   1:  PR[GP1:91,1] = PR[GP1:90,1] + 67.544;
   1:  PR[GP1:91,2] = PR[GP1:90,2] + 10.988;
   1:L PR[91] 10mm/sec CNT100;
   1:  PR[GP1:91,1] = PR[GP1:90,1] + 66.651;
   1:  PR[GP1:91,2] = PR[GP1:90,2] + 13.399;
   1:L PR[91] 10mm/sec CNT100;
   1:  PR[GP1:91,1] = PR[GP1:90,1] + 62.807;
   1:  PR[GP1:91,2] = PR[GP1:90,2] + 19.885;
   1:L PR[91] 10mm/sec CNT100;
   1:  PR[GP1:91,1] = PR[GP1:90,1] + 60.998;
   1:  PR[GP1:91,2] = PR[GP1:90,2] + 22.693;
   1:L PR[91] 10mm/sec CNT100;
   1:  PR[GP1:91,1] = PR[GP1:90,1] + 58.011;
   1:  PR[GP1:91,2] = PR[GP1:90,2] + 25.595;
   1:L PR[91] 10mm/sec CNT100;
   1:  PR[GP1:91,1] = PR[GP1:90,1] + 53.750;
   1:  PR[GP1:91,2] = PR[GP1:90,2] + 29.133;
   1:L PR[91] 10mm/sec CNT100;
   1:  PR[GP1:91,1] = PR[GP1:90,1] + 49.246;
   1:  PR[GP1:91,2] = PR[GP1:90,2] + 31.887;
   1:L PR[91] 10mm/sec CNT100;
   1:  PR[GP1:91,1] = PR[GP1:90,1] + 46.434;
   1:  PR[GP1:91,2] = PR[GP1:90,2] + 32.929;
   1:L PR[91] 10mm/sec CNT100;
   1:  PR[GP1:91,1] = PR[GP1:90,1] + 40.608;
   1:  PR[GP1:91,2] = PR[GP1:90,2] + 35.037;
   1:L PR[91] 10mm/sec CNT100;
   1:  PR[GP1:91,1] = PR[GP1:90,1] + 38.148;
   1:  PR[GP1:91,2] = PR[GP1:90,2] + 35.345;
   1:L PR[91] 10mm/sec CNT100;
   1:  PR[GP1:91,1] = PR[GP1:90,1] + 32.674;
   1:  PR[GP1:91,2] = PR[GP1:90,2] + 36.121;
   1:L PR[91] 10mm/sec CNT100;
   1:  PR[GP1:91,1] = PR[GP1:90,1] + 32.260;
   1:  PR[GP1:91,2] = PR[GP1:90,2] + 36.160;
   1:L PR[91] 10mm/sec CNT100;
   1:  PR[GP1:91,1] = PR[GP1:90,1] + 24.335;
   1:  PR[GP1:91,2] = PR[GP1:90,2] + 35.633;
   1:L PR[91] 10mm/sec CNT100;
   1:  PR[GP1:91,1] = PR[GP1:90,1] + 23.229;
   1:  PR[GP1:91,2] = PR[GP1:90,2] + 35.372;
   1:L PR[91] 10mm/sec CNT100;
   1:  PR[GP1:91,1] = PR[GP1:90,1] + 15.787;
   1:  PR[GP1:91,2] = PR[GP1:90,2] + 33.232;
   1:L PR[91] 10mm/sec CNT100;
   1:  PR[GP1:91,1] = PR[GP1:90,1] + 9.527;
   1:  PR[GP1:91,2] = PR[GP1:90,2] + 29.856;
   1:L PR[91] 10mm/sec CNT100;
   1:  PR[GP1:91,1] = PR[GP1:90,1] + 5.825;
   1:  PR[GP1:91,2] = PR[GP1:90,2] + 26.845;
   1:L PR[91] 10mm/sec CNT100;
   1:  PR[GP1:91,1] = PR[GP1:90,1] + 2.865;
   1:  PR[GP1:91,2] = PR[GP1:90,2] + 24.238;
   1:L PR[91] 10mm/sec CNT100;
   1:  PR[GP1:91,1] = PR[GP1:90,1] + 0.407;
   1:  PR[GP1:91,2] = PR[GP1:90,2] + 21.240;
   1:L PR[91] 10mm/sec CNT100;
   1:  PR[GP1:91,1] = PR[GP1:90,1] + -0.917;
   1:L PR[91] 10mm/sec CNT100;
   1:  PR[GP1:91,1] = PR[GP1:90,1] + -3.369;
   1:  PR[GP1:91,2] = PR[GP1:90,2] + 24.219;
   1:L PR[91] 10mm/sec CNT100;
   1:  PR[GP1:91,1] = PR[GP1:90,1] + -6.332;
   1:  PR[GP1:91,2] = PR[GP1:90,2] + 26.828;
   1:L PR[91] 10mm/sec CNT100;
   1:  PR[GP1:91,1] = PR[GP1:90,1] + -10.027;
   1:  PR[GP1:91,2] = PR[GP1:90,2] + 29.832;
   1:L PR[91] 10mm/sec CNT100;
   1:  PR[GP1:91,1] = PR[GP1:90,1] + -16.320;
   1:  PR[GP1:91,2] = PR[GP1:90,2] + 33.236;
   1:L PR[91] 10mm/sec CNT100;
   1:  PR[GP1:91,1] = PR[GP1:90,1] + -23.752;
   1:  PR[GP1:91,2] = PR[GP1:90,2] + 35.373;
   1:L PR[91] 10mm/sec CNT100;
   1:  PR[GP1:91,1] = PR[GP1:90,1] + -24.858;
   1:  PR[GP1:91,2] = PR[GP1:90,2] + 35.634;
   1:L PR[91] 10mm/sec CNT100;
   1:  PR[GP1:91,1] = PR[GP1:90,1] + -32.794;
   1:  PR[GP1:91,2] = PR[GP1:90,2] + 36.157;
   1:L PR[91] 10mm/sec CNT100;
   1:  PR[GP1:91,1] = PR[GP1:90,1] + -38.676;
   1:  PR[GP1:91,2] = PR[GP1:90,2] + 35.343;
   1:L PR[91] 10mm/sec CNT100;
   1:  PR[GP1:91,1] = PR[GP1:90,1] + -41.173;
   1:  PR[GP1:91,2] = PR[GP1:90,2] + 35.029;
   1:L PR[91] 10mm/sec CNT100;
   1:  PR[GP1:91,1] = PR[GP1:90,1] + -49.797;
   1:  PR[GP1:91,2] = PR[GP1:90,2] + 31.874;
   1:L PR[91] 10mm/sec CNT100;
   1:  PR[GP1:91,1] = PR[GP1:90,1] + -54.314;
   1:  PR[GP1:91,2] = PR[GP1:90,2] + 29.097;
   1:L PR[91] 10mm/sec CNT100;
   1:  PR[GP1:91,1] = PR[GP1:90,1] + -58.579;
   1:  PR[GP1:91,2] = PR[GP1:90,2] + 25.562;
   1:L PR[91] 10mm/sec CNT100;
   1:  PR[GP1:91,1] = PR[GP1:90,1] + -61.550;
   1:  PR[GP1:91,2] = PR[GP1:90,2] + 22.671;
   1:L PR[91] 10mm/sec CNT100;
   1:  PR[GP1:91,1] = PR[GP1:90,1] + -65.432;
   1:  PR[GP1:91,2] = PR[GP1:90,2] + 16.136;
   1:L PR[91] 10mm/sec CNT100;
   1:  PR[GP1:91,1] = PR[GP1:90,1] + -67.188;
   1:  PR[GP1:91,2] = PR[GP1:90,2] + 13.362;
   1:L PR[91] 10mm/sec CNT100;
   1:  PR[GP1:91,1] = PR[GP1:90,1] + -68.087;
   1:  PR[GP1:91,2] = PR[GP1:90,2] + 10.901;
   1:L PR[91] 10mm/sec CNT100;
   1:  PR[GP1:91,1] = PR[GP1:90,1] + -69.627;
   1:  PR[GP1:91,2] = PR[GP1:90,2] + 2.415;
   1:L PR[91] 10mm/sec CNT100;
   1:  PR[GP1:91,1] = PR[GP1:90,1] + -69.862;
   1:  PR[GP1:91,2] = PR[GP1:90,2] + 0.301;
   1:L PR[91] 10mm/sec CNT100;
   1:  PR[GP1:91,1] = PR[GP1:90,1] + -68.344;
   1:  PR[GP1:91,2] = PR[GP1:90,2] + -7.941;
   1:L PR[91] 10mm/sec CNT100;
   1:  PR[GP1:91,1] = PR[GP1:90,1] + -68.080;
   1:  PR[GP1:91,2] = PR[GP1:90,2] + -10.363;
   1:L PR[91] 10mm/sec CNT100;
   1:  PR[GP1:91,1] = PR[GP1:90,1] + -67.185;
   1:  PR[GP1:91,2] = PR[GP1:90,2] + -12.813;
   1:L PR[91] 10mm/sec CNT100;
   1:  PR[GP1:91,1] = PR[GP1:90,1] + -63.342;
   1:  PR[GP1:91,2] = PR[GP1:90,2] + -19.317;
   1:L PR[91] 10mm/sec CNT100;
   1:  PR[GP1:91,1] = PR[GP1:90,1] + -61.557;
   1:  PR[GP1:91,2] = PR[GP1:90,2] + -22.106;
   1:L PR[91] 10mm/sec CNT100;
   1:  PR[GP1:91,1] = PR[GP1:90,1] + -58.579;
   1:  PR[GP1:91,2] = PR[GP1:90,2] + -25.004;
   1:L PR[91] 10mm/sec CNT100;
   1:  PR[GP1:91,1] = PR[GP1:90,1] + -54.314;
   1:  PR[GP1:91,2] = PR[GP1:90,2] + -28.539;
   1:L PR[91] 10mm/sec CNT100;
   1:  PR[GP1:91,1] = PR[GP1:90,1] + -49.796;
   1:  PR[GP1:91,2] = PR[GP1:90,2] + -31.317;
   1:L PR[91] 10mm/sec CNT100;
   1:  PR[GP1:91,1] = PR[GP1:90,1] + -46.981;
   1:  PR[GP1:91,2] = PR[GP1:90,2] + -32.360;
   1:L PR[91] 10mm/sec CNT100;
   1:  PR[GP1:91,1] = PR[GP1:90,1] + -41.174;
   1:  PR[GP1:91,2] = PR[GP1:90,2] + -34.471;
   1:L PR[91] 10mm/sec CNT100;
   1:  PR[GP1:91,1] = PR[GP1:90,1] + -38.674;
   1:  PR[GP1:91,2] = PR[GP1:90,2] + -34.785;
   1:L PR[91] 10mm/sec CNT100;
   1:  PR[GP1:91,1] = PR[GP1:90,1] + -33.223;
   1:  PR[GP1:91,2] = PR[GP1:90,2] + -35.561;
   1:L PR[91] 10mm/sec CNT100;
   1:  PR[GP1:91,1] = PR[GP1:90,1] + -32.812;
   1:  PR[GP1:91,2] = PR[GP1:90,2] + -35.600;
   1:L PR[91] 10mm/sec CNT100;
   1:  PR[GP1:91,1] = PR[GP1:90,1] + -24.868;
   1:  PR[GP1:91,2] = PR[GP1:90,2] + -35.076;
   1:L PR[91] 10mm/sec CNT100;
   1:  PR[GP1:91,1] = PR[GP1:90,1] + -23.781;
   1:  PR[GP1:91,2] = PR[GP1:90,2] + -34.828;
   1:L PR[91] 10mm/sec CNT100;
   1:  PR[GP1:91,1] = PR[GP1:90,1] + -16.362;
   1:  PR[GP1:91,2] = PR[GP1:90,2] + -32.697;
   1:L PR[91] 10mm/sec CNT100;
   1:  PR[GP1:91,1] = PR[GP1:90,1] + -15.004;
   1:  PR[GP1:91,2] = PR[GP1:90,2] + -31.901;
   1:L PR[91] 10mm/sec CNT100;
   1:  PR[GP1:91,1] = PR[GP1:90,1] + -9.177;
   1:  PR[GP1:91,2] = PR[GP1:90,2] + -28.729;
   1:L PR[91] 10mm/sec CNT100;
   1:  PR[GP1:91,1] = PR[GP1:90,1] + -6.377;
   1:  PR[GP1:91,2] = PR[GP1:90,2] + -26.314;
   1:L PR[91] 10mm/sec CNT100;
   1:  PR[GP1:91,1] = PR[GP1:90,1] + -3.388;
   1:  PR[GP1:91,2] = PR[GP1:90,2] + -23.682;
   1:L PR[91] 10mm/sec CNT100;
   1:  PR[GP1:91,1] = PR[GP1:90,1] + -0.915;
   1:  PR[GP1:91,2] = PR[GP1:90,2] + -20.682;
   1:L PR[91] 10mm/sec CNT100;
   1:  PR[GP1:91,1] = PR[GP1:90,1] + 0.403;
   1:L PR[91] 10mm/sec CNT100;
   1:  PR[GP1:91,1] = PR[GP1:90,1] + 2.658;
   1:  PR[GP1:91,2] = PR[GP1:90,2] + -23.788;
   1:  PR[GP1:91,3] = PR[GP1:90,3] + 47.275;
   1:L PR[91] 10mm/sec CNT100;
   1:  PR[GP1:91,1] = PR[GP1:90,1] + 5.390;
   1:  PR[GP1:91,2] = PR[GP1:90,2] + -26.193;
   1:L PR[91] 10mm/sec CNT100;
   1:  PR[GP1:91,1] = PR[GP1:90,1] + 8.429;
   1:  PR[GP1:91,2] = PR[GP1:90,2] + -28.820;
   1:L PR[91] 10mm/sec CNT100;
   1:  PR[GP1:91,1] = PR[GP1:90,1] + 14.058;
   1:  PR[GP1:91,2] = PR[GP1:90,2] + -31.876;
   1:L PR[91] 10mm/sec CNT100;
   1:  PR[GP1:91,1] = PR[GP1:90,1] + 15.574;
   1:  PR[GP1:91,2] = PR[GP1:90,2] + -32.763;
   1:L PR[91] 10mm/sec CNT100;
   1:  PR[GP1:91,1] = PR[GP1:90,1] + 22.883;
   1:  PR[GP1:91,2] = PR[GP1:90,2] + -34.862;
   1:L PR[91] 10mm/sec CNT100;
   1:  PR[GP1:91,1] = PR[GP1:90,1] + 24.168;
   1:  PR[GP1:91,2] = PR[GP1:90,2] + -35.156;
   1:L PR[91] 10mm/sec CNT100;
   1:  PR[GP1:91,1] = PR[GP1:90,1] + 31.952;
   1:  PR[GP1:91,2] = PR[GP1:90,2] + -35.673;
   1:L PR[91] 10mm/sec CNT100;
   1:  PR[GP1:91,1] = PR[GP1:90,1] + 40.523;
   1:  PR[GP1:91,2] = PR[GP1:90,2] + -34.492;
   1:L PR[91] 10mm/sec CNT100;
   1:  PR[GP1:91,1] = PR[GP1:90,1] + 48.902;
   1:  PR[GP1:91,2] = PR[GP1:90,2] + -31.442;
   1:L PR[91] 10mm/sec CNT100;
   1:  PR[GP1:91,1] = PR[GP1:90,1] + 53.812;
   1:  PR[GP1:91,2] = PR[GP1:90,2] + -28.438;
   1:L PR[91] 10mm/sec CNT100;
   1:  PR[GP1:91,1] = PR[GP1:90,1] + 57.483;
   1:  PR[GP1:91,2] = PR[GP1:90,2] + -25.391;
   1:L PR[91] 10mm/sec CNT100;
   1:  PR[GP1:91,1] = PR[GP1:90,1] + 60.839;
   1:  PR[GP1:91,2] = PR[GP1:90,2] + -22.131;
   1:L PR[91] 10mm/sec CNT100;
   1:  PR[GP1:91,1] = PR[GP1:90,1] + 64.319;
   1:  PR[GP1:91,2] = PR[GP1:90,2] + -16.291;
   1:L PR[91] 10mm/sec CNT100;
   1:  PR[GP1:91,1] = PR[GP1:90,1] + 66.397;
   1:  PR[GP1:91,2] = PR[GP1:90,2] + -13.029;
   1:L PR[91] 10mm/sec CNT100;
   1:  PR[GP1:91,1] = PR[GP1:90,1] + 67.447;
   1:  PR[GP1:91,2] = PR[GP1:90,2] + -10.193;
   1:L PR[91] 10mm/sec CNT100;
   1:  PR[GP1:91,1] = PR[GP1:90,1] + 68.867;
   1:  PR[GP1:91,2] = PR[GP1:90,2] + -2.360;
   1:L PR[91] 10mm/sec CNT100;
   1:  PR[GP1:91,1] = PR[GP1:90,1] + 69.162;
   1:  PR[GP1:91,2] = PR[GP1:90,2] + 0.258;
   1:L PR[91] 10mm/sec CNT100;
   1:  PR[GP1:91,1] = PR[GP1:90,1] + 67.760;
   1:  PR[GP1:91,2] = PR[GP1:90,2] + 7.881;
   1:L PR[91] 10mm/sec CNT100;
   1:  PR[GP1:91,1] = PR[GP1:90,1] + 67.440;
   1:  PR[GP1:91,2] = PR[GP1:90,2] + 10.771;
   1:L PR[91] 10mm/sec CNT100;
   1:  PR[GP1:91,1] = PR[GP1:90,1] + 66.394;
   1:  PR[GP1:91,2] = PR[GP1:90,2] + 13.597;
   1:L PR[91] 10mm/sec CNT100;
   1:  PR[GP1:91,1] = PR[GP1:90,1] + 62.884;
   1:  PR[GP1:91,2] = PR[GP1:90,2] + 19.520;
   1:L PR[91] 10mm/sec CNT100;
   1:  PR[GP1:91,1] = PR[GP1:90,1] + 60.846;
   1:  PR[GP1:91,2] = PR[GP1:90,2] + 22.682;
   1:L PR[91] 10mm/sec CNT100;
   1:  PR[GP1:91,1] = PR[GP1:90,1] + 57.483;
   1:  PR[GP1:91,2] = PR[GP1:90,2] + 25.949;
   1:L PR[91] 10mm/sec CNT100;
   1:  PR[GP1:91,1] = PR[GP1:90,1] + 53.813;
   1:  PR[GP1:91,2] = PR[GP1:90,2] + 28.996;
   1:L PR[91] 10mm/sec CNT100;
   1:  PR[GP1:91,1] = PR[GP1:90,1] + 48.900;
   1:  PR[GP1:91,2] = PR[GP1:90,2] + 32.001;
   1:L PR[91] 10mm/sec CNT100;
   1:  PR[GP1:91,1] = PR[GP1:90,1] + 46.745;
   1:  PR[GP1:91,2] = PR[GP1:90,2] + 32.799;
   1:L PR[91] 10mm/sec CNT100;
   1:  PR[GP1:91,1] = PR[GP1:90,1] + 40.523;
   1:  PR[GP1:91,2] = PR[GP1:90,2] + 35.050;
   1:L PR[91] 10mm/sec CNT100;
   1:  PR[GP1:91,1] = PR[GP1:90,1] + 32.575;
   1:  PR[GP1:91,2] = PR[GP1:90,2] + 36.174;
   1:L PR[91] 10mm/sec CNT100;
   1:  PR[GP1:91,1] = PR[GP1:90,1] + 31.958;
   1:  PR[GP1:91,2] = PR[GP1:90,2] + 36.231;
   1:L PR[91] 10mm/sec CNT100;
   1:  PR[GP1:91,1] = PR[GP1:90,1] + 24.156;
   1:  PR[GP1:91,2] = PR[GP1:90,2] + 35.713;
   1:L PR[91] 10mm/sec CNT100;
   1:  PR[GP1:91,1] = PR[GP1:90,1] + 22.848;
   1:  PR[GP1:91,2] = PR[GP1:90,2] + 35.404;
   1:L PR[91] 10mm/sec CNT100;
   1:  PR[GP1:91,1] = PR[GP1:90,1] + 15.529;
   1:  PR[GP1:91,2] = PR[GP1:90,2] + 33.300;
   1:L PR[91] 10mm/sec CNT100;
   1:  PR[GP1:91,1] = PR[GP1:90,1] + 9.354;
   1:  PR[GP1:91,2] = PR[GP1:90,2] + 29.970;
   1:L PR[91] 10mm/sec CNT100;
   1:  PR[GP1:91,1] = PR[GP1:90,1] + 5.340;
   1:  PR[GP1:91,2] = PR[GP1:90,2] + 26.705;
   1:L PR[91] 10mm/sec CNT100;
   1:  PR[GP1:91,1] = PR[GP1:90,1] + 2.636;
   1:  PR[GP1:91,2] = PR[GP1:90,2] + 24.324;
   1:L PR[91] 10mm/sec CNT100;
   1:  PR[GP1:91,1] = PR[GP1:90,1] + 0.374;
   1:  PR[GP1:91,2] = PR[GP1:90,2] + 21.565;
   1:L PR[91] 10mm/sec CNT100;
   1:  PR[GP1:91,1] = PR[GP1:90,1] + -0.885;
   1:L PR[91] 10mm/sec CNT100;
   1:  PR[GP1:91,1] = PR[GP1:90,1] + -3.142;
   1:  PR[GP1:91,2] = PR[GP1:90,2] + 24.306;
   1:L PR[91] 10mm/sec CNT100;
   1:  PR[GP1:91,1] = PR[GP1:90,1] + -5.849;
   1:  PR[GP1:91,2] = PR[GP1:90,2] + 26.690;
   1:L PR[91] 10mm/sec CNT100;
   1:  PR[GP1:91,1] = PR[GP1:90,1] + -9.854;
   1:  PR[GP1:91,2] = PR[GP1:90,2] + 29.946;
   1:L PR[91] 10mm/sec CNT100;
   1:  PR[GP1:91,1] = PR[GP1:90,1] + -16.062;
   1:  PR[GP1:91,2] = PR[GP1:90,2] + 33.303;
   1:L PR[91] 10mm/sec CNT100;
   1:  PR[GP1:91,1] = PR[GP1:90,1] + -23.371;
   1:  PR[GP1:91,2] = PR[GP1:90,2] + 35.405;
   1:L PR[91] 10mm/sec CNT100;
   1:  PR[GP1:91,1] = PR[GP1:90,1] + -24.679;
   1:  PR[GP1:91,2] = PR[GP1:90,2] + 35.714;
   1:L PR[91] 10mm/sec CNT100;
   1:  PR[GP1:91,1] = PR[GP1:90,1] + -32.492;
   1:  PR[GP1:91,2] = PR[GP1:90,2] + 36.229;
   1:L PR[91] 10mm/sec CNT100;
   1:  PR[GP1:91,1] = PR[GP1:90,1] + -41.091;
   1:  PR[GP1:91,2] = PR[GP1:90,2] + 35.042;
   1:L PR[91] 10mm/sec CNT100;
   1:  PR[GP1:91,1] = PR[GP1:90,1] + -49.453;
   1:  PR[GP1:91,2] = PR[GP1:90,2] + 31.987;
   1:L PR[91] 10mm/sec CNT100;
   1:  PR[GP1:91,1] = PR[GP1:90,1] + -54.380;
   1:  PR[GP1:91,2] = PR[GP1:90,2] + 28.958;
   1:L PR[91] 10mm/sec CNT100;
   1:  PR[GP1:91,1] = PR[GP1:90,1] + -58.056;
   1:  PR[GP1:91,2] = PR[GP1:90,2] + 25.911;
   1:L PR[91] 10mm/sec CNT100;
   1:  PR[GP1:91,1] = PR[GP1:90,1] + -61.402;
   1:  PR[GP1:91,2] = PR[GP1:90,2] + 22.655;
   1:L PR[91] 10mm/sec CNT100;
   1:  PR[GP1:91,1] = PR[GP1:90,1] + -64.883;
   1:  PR[GP1:91,2] = PR[GP1:90,2] + 16.796;
   1:L PR[91] 10mm/sec CNT100;
   1:  PR[GP1:91,1] = PR[GP1:90,1] + -66.932;
   1:  PR[GP1:91,2] = PR[GP1:90,2] + 13.559;
   1:L PR[91] 10mm/sec CNT100;
   1:  PR[GP1:91,1] = PR[GP1:90,1] + -67.986;
   1:  PR[GP1:91,2] = PR[GP1:90,2] + 10.676;
   1:L PR[91] 10mm/sec CNT100;
   1:  PR[GP1:91,1] = PR[GP1:90,1] + -69.404;
   1:  PR[GP1:91,2] = PR[GP1:90,2] + 2.859;
   1:L PR[91] 10mm/sec CNT100;
   1:  PR[GP1:91,1] = PR[GP1:90,1] + -69.689;
   1:  PR[GP1:91,2] = PR[GP1:90,2] + 0.301;
   1:L PR[91] 10mm/sec CNT100;
   1:  PR[GP1:91,1] = PR[GP1:90,1] + -68.287;
   1:  PR[GP1:91,2] = PR[GP1:90,2] + -7.309;
   1:L PR[91] 10mm/sec CNT100;
   1:  PR[GP1:91,1] = PR[GP1:90,1] + -67.978;
   1:  PR[GP1:91,2] = PR[GP1:90,2] + -10.138;
   1:L PR[91] 10mm/sec CNT100;
   1:  PR[GP1:91,1] = PR[GP1:90,1] + -66.929;
   1:  PR[GP1:91,2] = PR[GP1:90,2] + -13.010;
   1:L PR[91] 10mm/sec CNT100;
   1:  PR[GP1:91,1] = PR[GP1:90,1] + -63.419;
   1:  PR[GP1:91,2] = PR[GP1:90,2] + -18.950;
   1:L PR[91] 10mm/sec CNT100;
   1:  PR[GP1:91,1] = PR[GP1:90,1] + -61.409;
   1:  PR[GP1:91,2] = PR[GP1:90,2] + -22.090;
   1:L PR[91] 10mm/sec CNT100;
   1:  PR[GP1:91,1] = PR[GP1:90,1] + -58.056;
   1:  PR[GP1:91,2] = PR[GP1:90,2] + -25.353;
   1:L PR[91] 10mm/sec CNT100;
   1:  PR[GP1:91,1] = PR[GP1:90,1] + -54.380;
   1:  PR[GP1:91,2] = PR[GP1:90,2] + -28.400;
   1:L PR[91] 10mm/sec CNT100;
   1:  PR[GP1:91,1] = PR[GP1:90,1] + -49.452;
   1:  PR[GP1:91,2] = PR[GP1:90,2] + -31.430;
   1:L PR[91] 10mm/sec CNT100;
   1:  PR[GP1:91,1] = PR[GP1:90,1] + -47.293;
   1:  PR[GP1:91,2] = PR[GP1:90,2] + -32.230;
   1:L PR[91] 10mm/sec CNT100;
   1:  PR[GP1:91,1] = PR[GP1:90,1] + -41.091;
   1:  PR[GP1:91,2] = PR[GP1:90,2] + -34.484;
   1:L PR[91] 10mm/sec CNT100;
   1:  PR[GP1:91,1] = PR[GP1:90,1] + -33.126;
   1:  PR[GP1:91,2] = PR[GP1:90,2] + -35.614;
   1:L PR[91] 10mm/sec CNT100;
   1:  PR[GP1:91,1] = PR[GP1:90,1] + -32.512;
   1:  PR[GP1:91,2] = PR[GP1:90,2] + -35.672;
   1:L PR[91] 10mm/sec CNT100;
   1:  PR[GP1:91,1] = PR[GP1:90,1] + -24.691;
   1:  PR[GP1:91,2] = PR[GP1:90,2] + -35.156;
   1:L PR[91] 10mm/sec CNT100;
   1:  PR[GP1:91,1] = PR[GP1:90,1] + -23.406;
   1:  PR[GP1:91,2] = PR[GP1:90,2] + -34.862;
   1:L PR[91] 10mm/sec CNT100;
   1:  PR[GP1:91,1] = PR[GP1:90,1] + -16.107;
   1:  PR[GP1:91,2] = PR[GP1:90,2] + -32.766;
   1:L PR[91] 10mm/sec CNT100;
   1:  PR[GP1:91,1] = PR[GP1:90,1] + -14.593;
   1:  PR[GP1:91,2] = PR[GP1:90,2] + -31.879;
   1:L PR[91] 10mm/sec CNT100;
   1:  PR[GP1:91,1] = PR[GP1:90,1] + -8.933;
   1:  PR[GP1:91,2] = PR[GP1:90,2] + -28.798;
   1:L PR[91] 10mm/sec CNT100;
   1:  PR[GP1:91,1] = PR[GP1:90,1] + -5.897;
   1:  PR[GP1:91,2] = PR[GP1:90,2] + -26.179;
   1:L PR[91] 10mm/sec CNT100;
   1:  PR[GP1:91,1] = PR[GP1:90,1] + -3.162;
   1:  PR[GP1:91,2] = PR[GP1:90,2] + -23.771;
   1:L PR[91] 10mm/sec CNT100;
   1:  PR[GP1:91,1] = PR[GP1:90,1] + -0.884;
   1:  PR[GP1:91,2] = PR[GP1:90,2] + -21.007;
   1:L PR[91] 10mm/sec CNT100;
   1:  PR[GP1:91,1] = PR[GP1:90,1] + 0.371;
   1:L PR[91] 10mm/sec CNT100;
   1:  PR[GP1:91,1] = PR[GP1:90,1] + 2.431;
   1:  PR[GP1:91,2] = PR[GP1:90,2] + -23.875;
   1:  PR[GP1:91,3] = PR[GP1:90,3] + 47.885;
   1:L PR[91] 10mm/sec CNT100;
   1:  PR[GP1:91,1] = PR[GP1:90,1] + 4.909;
   1:  PR[GP1:91,2] = PR[GP1:90,2] + -26.057;
   1:L PR[91] 10mm/sec CNT100;
   1:  PR[GP1:91,1] = PR[GP1:90,1] + 8.185;
   1:  PR[GP1:91,2] = PR[GP1:90,2] + -28.889;
   1:L PR[91] 10mm/sec CNT100;
   1:  PR[GP1:91,1] = PR[GP1:90,1] + 13.648;
   1:  PR[GP1:91,2] = PR[GP1:90,2] + -31.854;
   1:L PR[91] 10mm/sec CNT100;
   1:  PR[GP1:91,1] = PR[GP1:90,1] + 15.319;
   1:  PR[GP1:91,2] = PR[GP1:90,2] + -32.832;
   1:L PR[91] 10mm/sec CNT100;
   1:  PR[GP1:91,1] = PR[GP1:90,1] + 22.507;
   1:  PR[GP1:91,2] = PR[GP1:90,2] + -34.896;
   1:L PR[91] 10mm/sec CNT100;
   1:  PR[GP1:91,1] = PR[GP1:90,1] + 23.991;
   1:  PR[GP1:91,2] = PR[GP1:90,2] + -35.236;
   1:L PR[91] 10mm/sec CNT100;
   1:  PR[GP1:91,1] = PR[GP1:90,1] + 31.652;
   1:  PR[GP1:91,2] = PR[GP1:90,2] + -35.745;
   1:L PR[91] 10mm/sec CNT100;
   1:  PR[GP1:91,1] = PR[GP1:90,1] + 40.318;
   1:  PR[GP1:91,2] = PR[GP1:90,2] + -34.557;
   1:L PR[91] 10mm/sec CNT100;
   1:  PR[GP1:91,1] = PR[GP1:90,1] + 48.556;
   1:  PR[GP1:91,2] = PR[GP1:90,2] + -31.556;
   1:L PR[91] 10mm/sec CNT100;
   1:  PR[GP1:91,1] = PR[GP1:90,1] + 53.875;
   1:  PR[GP1:91,2] = PR[GP1:90,2] + -28.302;
   1:L PR[91] 10mm/sec CNT100;
   1:  PR[GP1:91,1] = PR[GP1:90,1] + 56.955;
   1:  PR[GP1:91,2] = PR[GP1:90,2] + -25.745;
   1:L PR[91] 10mm/sec CNT100;
   1:  PR[GP1:91,1] = PR[GP1:90,1] + 60.687;
   1:  PR[GP1:91,2] = PR[GP1:90,2] + -22.120;
   1:L PR[91] 10mm/sec CNT100;
   1:  PR[GP1:91,1] = PR[GP1:90,1] + 63.765;
   1:  PR[GP1:91,2] = PR[GP1:90,2] + -16.956;
   1:L PR[91] 10mm/sec CNT100;
   1:  PR[GP1:91,1] = PR[GP1:90,1] + 66.140;
   1:  PR[GP1:91,2] = PR[GP1:90,2] + -13.227;
   1:L PR[91] 10mm/sec CNT100;
   1:  PR[GP1:91,1] = PR[GP1:90,1] + 67.344;
   1:  PR[GP1:91,2] = PR[GP1:90,2] + -9.976;
   1:L PR[91] 10mm/sec CNT100;
   1:  PR[GP1:91,1] = PR[GP1:90,1] + 68.641;
   1:  PR[GP1:91,2] = PR[GP1:90,2] + -2.814;
   1:L PR[91] 10mm/sec CNT100;
   1:  PR[GP1:91,1] = PR[GP1:90,1] + 68.988;
   1:  PR[GP1:91,2] = PR[GP1:90,2] + 0.258;
   1:L PR[91] 10mm/sec CNT100;
   1:  PR[GP1:91,1] = PR[GP1:90,1] + 67.703;
   1:  PR[GP1:91,2] = PR[GP1:90,2] + 7.248;
   1:L PR[91] 10mm/sec CNT100;
   1:  PR[GP1:91,1] = PR[GP1:90,1] + 67.337;
   1:  PR[GP1:91,2] = PR[GP1:90,2] + 10.553;
   1:L PR[91] 10mm/sec CNT100;
   1:  PR[GP1:91,1] = PR[GP1:90,1] + 66.136;
   1:  PR[GP1:91,2] = PR[GP1:90,2] + 13.795;
   1:L PR[91] 10mm/sec CNT100;
   1:  PR[GP1:91,1] = PR[GP1:90,1] + 62.960;
   1:  PR[GP1:91,2] = PR[GP1:90,2] + 19.154;
   1:L PR[91] 10mm/sec CNT100;
   1:  PR[GP1:91,1] = PR[GP1:90,1] + 60.695;
   1:  PR[GP1:91,2] = PR[GP1:90,2] + 22.670;
   1:L PR[91] 10mm/sec CNT100;
   1:  PR[GP1:91,1] = PR[GP1:90,1] + 56.955;
   1:  PR[GP1:91,2] = PR[GP1:90,2] + 26.303;
   1:L PR[91] 10mm/sec CNT100;
   1:  PR[GP1:91,1] = PR[GP1:90,1] + 53.875;
   1:  PR[GP1:91,2] = PR[GP1:90,2] + 28.860;
   1:L PR[91] 10mm/sec CNT100;
   1:  PR[GP1:91,1] = PR[GP1:90,1] + 48.556;
   1:  PR[GP1:91,2] = PR[GP1:90,2] + 32.114;
   1:L PR[91] 10mm/sec CNT100;
   1:  PR[GP1:91,1] = PR[GP1:90,1] + 40.315;
   1:  PR[GP1:91,2] = PR[GP1:90,2] + 35.116;
   1:L PR[91] 10mm/sec CNT100;
   1:  PR[GP1:91,1] = PR[GP1:90,1] + 32.476;
   1:  PR[GP1:91,2] = PR[GP1:90,2] + 36.227;
   1:L PR[91] 10mm/sec CNT100;
   1:  PR[GP1:91,1] = PR[GP1:90,1] + 31.655;
   1:  PR[GP1:91,2] = PR[GP1:90,2] + 36.303;
   1:L PR[91] 10mm/sec CNT100;
   1:  PR[GP1:91,1] = PR[GP1:90,1] + 23.977;
   1:  PR[GP1:91,2] = PR[GP1:90,2] + 35.793;
   1:L PR[91] 10mm/sec CNT100;
   1:  PR[GP1:91,1] = PR[GP1:90,1] + 22.468;
   1:  PR[GP1:91,2] = PR[GP1:90,2] + 35.437;
   1:L PR[91] 10mm/sec CNT100;
   1:  PR[GP1:91,1] = PR[GP1:90,1] + 15.271;
   1:  PR[GP1:91,2] = PR[GP1:90,2] + 33.368;
   1:L PR[91] 10mm/sec CNT100;
   1:  PR[GP1:91,1] = PR[GP1:90,1] + 9.182;
   1:  PR[GP1:91,2] = PR[GP1:90,2] + 30.084;
   1:L PR[91] 10mm/sec CNT100;
   1:  PR[GP1:91,1] = PR[GP1:90,1] + 4.855;
   1:  PR[GP1:91,2] = PR[GP1:90,2] + 26.566;
   1:L PR[91] 10mm/sec CNT100;
   1:  PR[GP1:91,1] = PR[GP1:90,1] + 2.407;
   1:  PR[GP1:91,2] = PR[GP1:90,2] + 24.409;
   1:L PR[91] 10mm/sec CNT100;
   1:  PR[GP1:91,1] = PR[GP1:90,1] + 0.341;
   1:  PR[GP1:91,2] = PR[GP1:90,2] + 21.890;
   1:L PR[91] 10mm/sec CNT100;
   1:  PR[GP1:91,1] = PR[GP1:90,1] + -0.854;
   1:L PR[91] 10mm/sec CNT100;
   1:  PR[GP1:91,1] = PR[GP1:90,1] + -2.914;
   1:  PR[GP1:91,2] = PR[GP1:90,2] + 24.393;
   1:L PR[91] 10mm/sec CNT100;
   1:  PR[GP1:91,1] = PR[GP1:90,1] + -5.366;
   1:  PR[GP1:91,2] = PR[GP1:90,2] + 26.552;
   1:L PR[91] 10mm/sec CNT100;
   1:  PR[GP1:91,1] = PR[GP1:90,1] + -9.682;
   1:  PR[GP1:91,2] = PR[GP1:90,2] + 30.061;
   1:L PR[91] 10mm/sec CNT100;
   1:  PR[GP1:91,1] = PR[GP1:90,1] + -15.803;
   1:  PR[GP1:91,2] = PR[GP1:90,2] + 33.371;
   1:L PR[91] 10mm/sec CNT100;
   1:  PR[GP1:91,1] = PR[GP1:90,1] + -22.990;
   1:  PR[GP1:91,2] = PR[GP1:90,2] + 35.437;
   1:L PR[91] 10mm/sec CNT100;
   1:  PR[GP1:91,1] = PR[GP1:90,1] + -24.500;
   1:  PR[GP1:91,2] = PR[GP1:90,2] + 35.794;
   1:L PR[91] 10mm/sec CNT100;
   1:  PR[GP1:91,1] = PR[GP1:90,1] + -32.189;
   1:  PR[GP1:91,2] = PR[GP1:90,2] + 36.301;
   1:L PR[91] 10mm/sec CNT100;
   1:  PR[GP1:91,1] = PR[GP1:90,1] + -40.886;
   1:  PR[GP1:91,2] = PR[GP1:90,2] + 35.106;
   1:L PR[91] 10mm/sec CNT100;
   1:  PR[GP1:91,1] = PR[GP1:90,1] + -49.109;
   1:  PR[GP1:91,2] = PR[GP1:90,2] + 32.100;
   1:L PR[91] 10mm/sec CNT100;
   1:  PR[GP1:91,1] = PR[GP1:90,1] + -54.446;
   1:  PR[GP1:91,2] = PR[GP1:90,2] + 28.819;
   1:L PR[91] 10mm/sec CNT100;
   1:  PR[GP1:91,1] = PR[GP1:90,1] + -57.533;
   1:  PR[GP1:91,2] = PR[GP1:90,2] + 26.260;
   1:L PR[91] 10mm/sec CNT100;
   1:  PR[GP1:91,1] = PR[GP1:90,1] + -61.254;
   1:  PR[GP1:91,2] = PR[GP1:90,2] + 22.640;
   1:L PR[91] 10mm/sec CNT100;
   1:  PR[GP1:91,1] = PR[GP1:90,1] + -64.334;
   1:  PR[GP1:91,2] = PR[GP1:90,2] + 17.456;
   1:L PR[91] 10mm/sec CNT100;
   1:  PR[GP1:91,1] = PR[GP1:90,1] + -66.676;
   1:  PR[GP1:91,2] = PR[GP1:90,2] + 13.756;
   1:L PR[91] 10mm/sec CNT100;
   1:  PR[GP1:91,1] = PR[GP1:90,1] + -67.884;
   1:  PR[GP1:91,2] = PR[GP1:90,2] + 10.450;
   1:L PR[91] 10mm/sec CNT100;
   1:  PR[GP1:91,1] = PR[GP1:90,1] + -69.181;
   1:  PR[GP1:91,2] = PR[GP1:90,2] + 3.302;
   1:L PR[91] 10mm/sec CNT100;
   1:  PR[GP1:91,1] = PR[GP1:90,1] + -69.515;
   1:  PR[GP1:91,2] = PR[GP1:90,2] + 0.301;
   1:L PR[91] 10mm/sec CNT100;
   1:  PR[GP1:91,1] = PR[GP1:90,1] + -68.229;
   1:  PR[GP1:91,2] = PR[GP1:90,2] + -6.678;
   1:L PR[91] 10mm/sec CNT100;
   1:  PR[GP1:91,1] = PR[GP1:90,1] + -67.876;
   1:  PR[GP1:91,2] = PR[GP1:90,2] + -9.912;
   1:L PR[91] 10mm/sec CNT100;
   1:  PR[GP1:91,1] = PR[GP1:90,1] + -66.673;
   1:  PR[GP1:91,2] = PR[GP1:90,2] + -13.206;
   1:L PR[91] 10mm/sec CNT100;
   1:  PR[GP1:91,1] = PR[GP1:90,1] + -63.497;
   1:  PR[GP1:91,2] = PR[GP1:90,2] + -18.582;
   1:L PR[91] 10mm/sec CNT100;
   1:  PR[GP1:91,1] = PR[GP1:90,1] + -61.262;
   1:  PR[GP1:91,2] = PR[GP1:90,2] + -22.074;
   1:L PR[91] 10mm/sec CNT100;
   1:  PR[GP1:91,1] = PR[GP1:90,1] + -57.533;
   1:  PR[GP1:91,2] = PR[GP1:90,2] + -25.702;
   1:L PR[91] 10mm/sec CNT100;
   1:  PR[GP1:91,1] = PR[GP1:90,1] + -54.446;
   1:  PR[GP1:91,2] = PR[GP1:90,2] + -28.261;
   1:L PR[91] 10mm/sec CNT100;
   1:  PR[GP1:91,1] = PR[GP1:90,1] + -49.109;
   1:  PR[GP1:91,2] = PR[GP1:90,2] + -31.542;
   1:L PR[91] 10mm/sec CNT100;
   1:  PR[GP1:91,1] = PR[GP1:90,1] + -40.887;
   1:  PR[GP1:91,2] = PR[GP1:90,2] + -34.548;
   1:L PR[91] 10mm/sec CNT100;
   1:  PR[GP1:91,1] = PR[GP1:90,1] + -33.028;
   1:  PR[GP1:91,2] = PR[GP1:90,2] + -35.666;
   1:L PR[91] 10mm/sec CNT100;
   1:  PR[GP1:91,1] = PR[GP1:90,1] + -32.211;
   1:  PR[GP1:91,2] = PR[GP1:90,2] + -35.744;
   1:L PR[91] 10mm/sec CNT100;
   1:  PR[GP1:91,1] = PR[GP1:90,1] + -24.515;
   1:  PR[GP1:91,2] = PR[GP1:90,2] + -35.237;
   1:L PR[91] 10mm/sec CNT100;
   1:  PR[GP1:91,1] = PR[GP1:90,1] + -23.031;
   1:  PR[GP1:91,2] = PR[GP1:90,2] + -34.897;
   1:L PR[91] 10mm/sec CNT100;
   1:  PR[GP1:91,1] = PR[GP1:90,1] + -15.852;
   1:  PR[GP1:91,2] = PR[GP1:90,2] + -32.836;
   1:L PR[91] 10mm/sec CNT100;
   1:  PR[GP1:91,1] = PR[GP1:90,1] + -14.182;
   1:  PR[GP1:91,2] = PR[GP1:90,2] + -31.857;
   1:L PR[91] 10mm/sec CNT100;
   1:  PR[GP1:91,1] = PR[GP1:90,1] + -8.689;
   1:  PR[GP1:91,2] = PR[GP1:90,2] + -28.867;
   1:L PR[91] 10mm/sec CNT100;
   1:  PR[GP1:91,1] = PR[GP1:90,1] + -5.417;
   1:  PR[GP1:91,2] = PR[GP1:90,2] + -26.044;
   1:L PR[91] 10mm/sec CNT100;
   1:  PR[GP1:91,1] = PR[GP1:90,1] + -2.936;
   1:  PR[GP1:91,2] = PR[GP1:90,2] + -23.859;
   1:L PR[91] 10mm/sec CNT100;
   1:  PR[GP1:91,1] = PR[GP1:90,1] + -0.853;
   1:  PR[GP1:91,2] = PR[GP1:90,2] + -21.332;
   1:L PR[91] 10mm/sec CNT100;
   1:  PR[GP1:91,1] = PR[GP1:90,1] + 0.339;
   1:L PR[91] 10mm/sec CNT100;
   1:  PR[GP1:91,1] = PR[GP1:90,1] + 2.203;
   1:  PR[GP1:91,2] = PR[GP1:90,2] + -23.962;
   1:  PR[GP1:91,3] = PR[GP1:90,3] + 48.495;
   1:L PR[91] 10mm/sec CNT100;
   1:  PR[GP1:91,1] = PR[GP1:90,1] + 4.427;
   1:  PR[GP1:91,2] = PR[GP1:90,2] + -25.921;
   1:L PR[91] 10mm/sec CNT100;
   1:  PR[GP1:91,1] = PR[GP1:90,1] + 7.941;
   1:  PR[GP1:91,2] = PR[GP1:90,2] + -28.957;
   1:L PR[91] 10mm/sec CNT100;
   1:  PR[GP1:91,1] = PR[GP1:90,1] + 13.237;
   1:  PR[GP1:91,2] = PR[GP1:90,2] + -31.832;
   1:L PR[91] 10mm/sec CNT100;
   1:  PR[GP1:91,1] = PR[GP1:90,1] + 15.065;
   1:  PR[GP1:91,2] = PR[GP1:90,2] + -32.902;
   1:L PR[91] 10mm/sec CNT100;
   1:  PR[GP1:91,1] = PR[GP1:90,1] + 22.132;
   1:  PR[GP1:91,2] = PR[GP1:90,2] + -34.931;
   1:L PR[91] 10mm/sec CNT100;
   1:  PR[GP1:91,1] = PR[GP1:90,1] + 23.814;
   1:  PR[GP1:91,2] = PR[GP1:90,2] + -35.316;
   1:L PR[91] 10mm/sec CNT100;
   1:  PR[GP1:91,1] = PR[GP1:90,1] + 31.352;
   1:  PR[GP1:91,2] = PR[GP1:90,2] + -35.817;
   1:L PR[91] 10mm/sec CNT100;
   1:  PR[GP1:91,1] = PR[GP1:90,1] + 39.758;
   1:  PR[GP1:91,2] = PR[GP1:90,2] + -34.657;
   1:L PR[91] 10mm/sec CNT100;
   1:  PR[GP1:91,1] = PR[GP1:90,1] + 40.112;
   1:  PR[GP1:91,2] = PR[GP1:90,2] + -34.622;
   1:L PR[91] 10mm/sec CNT100;
   1:  PR[GP1:91,1] = PR[GP1:90,1] + 48.209;
   1:  PR[GP1:91,2] = PR[GP1:90,2] + -31.670;
   1:L PR[91] 10mm/sec CNT100;
   1:  PR[GP1:91,1] = PR[GP1:90,1] + 53.938;
   1:  PR[GP1:91,2] = PR[GP1:90,2] + -28.166;
   1:L PR[91] 10mm/sec CNT100;
   1:  PR[GP1:91,1] = PR[GP1:90,1] + 56.427;
   1:  PR[GP1:91,2] = PR[GP1:90,2] + -26.099;
   1:L PR[91] 10mm/sec CNT100;
   1:  PR[GP1:91,1] = PR[GP1:90,1] + 60.535;
   1:  PR[GP1:91,2] = PR[GP1:90,2] + -22.108;
   1:L PR[91] 10mm/sec CNT100;
   1:  PR[GP1:91,1] = PR[GP1:90,1] + 63.210;
   1:  PR[GP1:91,2] = PR[GP1:90,2] + -17.621;
   1:L PR[91] 10mm/sec CNT100;
   1:  PR[GP1:91,1] = PR[GP1:90,1] + 65.882;
   1:  PR[GP1:91,2] = PR[GP1:90,2] + -13.425;
   1:L PR[91] 10mm/sec CNT100;
   1:  PR[GP1:91,1] = PR[GP1:90,1] + 67.240;
   1:  PR[GP1:91,2] = PR[GP1:90,2] + -9.758;
   1:L PR[91] 10mm/sec CNT100;
   1:  PR[GP1:91,1] = PR[GP1:90,1] + 68.416;
   1:  PR[GP1:91,2] = PR[GP1:90,2] + -3.267;
   1:L PR[91] 10mm/sec CNT100;
   1:  PR[GP1:91,1] = PR[GP1:90,1] + 68.814;
   1:  PR[GP1:91,2] = PR[GP1:90,2] + 0.258;
   1:L PR[91] 10mm/sec CNT100;
   1:  PR[GP1:91,1] = PR[GP1:90,1] + 67.645;
   1:  PR[GP1:91,2] = PR[GP1:90,2] + 6.615;
   1:L PR[91] 10mm/sec CNT100;
   1:  PR[GP1:91,1] = PR[GP1:90,1] + 67.233;
   1:  PR[GP1:91,2] = PR[GP1:90,2] + 10.336;
   1:L PR[91] 10mm/sec CNT100;
   1:  PR[GP1:91,1] = PR[GP1:90,1] + 65.879;
   1:  PR[GP1:91,2] = PR[GP1:90,2] + 13.993;
   1:L PR[91] 10mm/sec CNT100;
   1:  PR[GP1:91,1] = PR[GP1:90,1] + 63.037;
   1:  PR[GP1:91,2] = PR[GP1:90,2] + 18.789;
   1:L PR[91] 10mm/sec CNT100;
   1:  PR[GP1:91,1] = PR[GP1:90,1] + 60.543;
   1:  PR[GP1:91,2] = PR[GP1:90,2] + 22.659;
   1:L PR[91] 10mm/sec CNT100;
   1:  PR[GP1:91,1] = PR[GP1:90,1] + 56.427;
   1:  PR[GP1:91,2] = PR[GP1:90,2] + 26.657;
   1:L PR[91] 10mm/sec CNT100;
   1:  PR[GP1:91,1] = PR[GP1:90,1] + 53.938;
   1:  PR[GP1:91,2] = PR[GP1:90,2] + 28.724;
   1:L PR[91] 10mm/sec CNT100;
   1:  PR[GP1:91,1] = PR[GP1:90,1] + 48.209;
   1:  PR[GP1:91,2] = PR[GP1:90,2] + 32.228;
   1:L PR[91] 10mm/sec CNT100;
   1:  PR[GP1:91,1] = PR[GP1:90,1] + 40.096;
   1:  PR[GP1:91,2] = PR[GP1:90,2] + 35.186;
   1:L PR[91] 10mm/sec CNT100;
   1:  PR[GP1:91,1] = PR[GP1:90,1] + 32.377;
   1:  PR[GP1:91,2] = PR[GP1:90,2] + 36.280;
   1:L PR[91] 10mm/sec CNT100;
   1:  PR[GP1:91,1] = PR[GP1:90,1] + 31.353;
   1:  PR[GP1:91,2] = PR[GP1:90,2] + 36.375;
   1:L PR[91] 10mm/sec CNT100;
   1:  PR[GP1:91,1] = PR[GP1:90,1] + 23.798;
   1:  PR[GP1:91,2] = PR[GP1:90,2] + 35.873;
   1:L PR[91] 10mm/sec CNT100;
   1:  PR[GP1:91,1] = PR[GP1:90,1] + 22.087;
   1:  PR[GP1:91,2] = PR[GP1:90,2] + 35.469;
   1:L PR[91] 10mm/sec CNT100;
   1:  PR[GP1:91,1] = PR[GP1:90,1] + 15.013;
   1:  PR[GP1:91,2] = PR[GP1:90,2] + 33.435;
   1:L PR[91] 10mm/sec CNT100;
   1:  PR[GP1:91,1] = PR[GP1:90,1] + 9.009;
   1:  PR[GP1:91,2] = PR[GP1:90,2] + 30.198;
   1:L PR[91] 10mm/sec CNT100;
   1:  PR[GP1:91,1] = PR[GP1:90,1] + 4.371;
   1:  PR[GP1:91,2] = PR[GP1:90,2] + 26.426;
   1:L PR[91] 10mm/sec CNT100;
   1:  PR[GP1:91,1] = PR[GP1:90,1] + 2.178;
   1:  PR[GP1:91,2] = PR[GP1:90,2] + 24.495;
   1:L PR[91] 10mm/sec CNT100;
   1:  PR[GP1:91,1] = PR[GP1:90,1] + 0.308;
   1:  PR[GP1:91,2] = PR[GP1:90,2] + 22.215;
   1:L PR[91] 10mm/sec CNT100;
   1:  PR[GP1:91,1] = PR[GP1:90,1] + -0.822;
   1:L PR[91] 10mm/sec CNT100;
   1:  PR[GP1:91,1] = PR[GP1:90,1] + -2.687;
   1:  PR[GP1:91,2] = PR[GP1:90,2] + 24.481;
   1:L PR[91] 10mm/sec CNT100;
   1:  PR[GP1:91,1] = PR[GP1:90,1] + -4.883;
   1:  PR[GP1:91,2] = PR[GP1:90,2] + 26.414;
   1:L PR[91] 10mm/sec CNT100;
   1:  PR[GP1:91,1] = PR[GP1:90,1] + -9.509;
   1:  PR[GP1:91,2] = PR[GP1:90,2] + 30.175;
   1:L PR[91] 10mm/sec CNT100;
   1:  PR[GP1:91,1] = PR[GP1:90,1] + -15.545;
   1:  PR[GP1:91,2] = PR[GP1:90,2] + 33.439;
   1:L PR[91] 10mm/sec CNT100;
   1:  PR[GP1:91,1] = PR[GP1:90,1] + -22.610;
   1:  PR[GP1:91,2] = PR[GP1:90,2] + 35.470;
   1:L PR[91] 10mm/sec CNT100;
   1:  PR[GP1:91,1] = PR[GP1:90,1] + -24.321;
   1:  PR[GP1:91,2] = PR[GP1:90,2] + 35.874;
   1:L PR[91] 10mm/sec CNT100;
   1:  PR[GP1:91,1] = PR[GP1:90,1] + -31.886;
   1:  PR[GP1:91,2] = PR[GP1:90,2] + 36.373;
   1:L PR[91] 10mm/sec CNT100;
   1:  PR[GP1:91,1] = PR[GP1:90,1] + -40.327;
   1:  PR[GP1:91,2] = PR[GP1:90,2] + 35.205;
   1:L PR[91] 10mm/sec CNT100;
   1:  PR[GP1:91,1] = PR[GP1:90,1] + -40.679;
   1:  PR[GP1:91,2] = PR[GP1:90,2] + 35.172;
   1:L PR[91] 10mm/sec CNT100;
   1:  PR[GP1:91,1] = PR[GP1:90,1] + -48.765;
   1:  PR[GP1:91,2] = PR[GP1:90,2] + 32.214;
   1:L PR[91] 10mm/sec CNT100;
   1:  PR[GP1:91,1] = PR[GP1:90,1] + -54.512;
   1:  PR[GP1:91,2] = PR[GP1:90,2] + 28.680;
   1:L PR[91] 10mm/sec CNT100;
   1:  PR[GP1:91,1] = PR[GP1:90,1] + -57.010;
   1:  PR[GP1:91,2] = PR[GP1:90,2] + 26.609;
   1:L PR[91] 10mm/sec CNT100;
   1:  PR[GP1:91,1] = PR[GP1:90,1] + -61.106;
   1:  PR[GP1:91,2] = PR[GP1:90,2] + 22.624;
   1:L PR[91] 10mm/sec CNT100;
   1:  PR[GP1:91,1] = PR[GP1:90,1] + -63.784;
   1:  PR[GP1:91,2] = PR[GP1:90,2] + 18.117;
   1:L PR[91] 10mm/sec CNT100;
   1:  PR[GP1:91,1] = PR[GP1:90,1] + -66.420;
   1:  PR[GP1:91,2] = PR[GP1:90,2] + 13.952;
   1:L PR[91] 10mm/sec CNT100;
   1:  PR[GP1:91,1] = PR[GP1:90,1] + -67.782;
   1:  PR[GP1:91,2] = PR[GP1:90,2] + 10.225;
   1:L PR[91] 10mm/sec CNT100;
   1:  PR[GP1:91,1] = PR[GP1:90,1] + -68.957;
   1:  PR[GP1:91,2] = PR[GP1:90,2] + 3.746;
   1:L PR[91] 10mm/sec CNT100;
   1:  PR[GP1:91,1] = PR[GP1:90,1] + -69.341;
   1:  PR[GP1:91,2] = PR[GP1:90,2] + 0.301;
   1:L PR[91] 10mm/sec CNT100;
   1:  PR[GP1:91,1] = PR[GP1:90,1] + -68.172;
   1:  PR[GP1:91,2] = PR[GP1:90,2] + -6.046;
   1:L PR[91] 10mm/sec CNT100;
   1:  PR[GP1:91,1] = PR[GP1:90,1] + -67.774;
   1:  PR[GP1:91,2] = PR[GP1:90,2] + -9.687;
   1:L PR[91] 10mm/sec CNT100;
   1:  PR[GP1:91,1] = PR[GP1:90,1] + -66.416;
   1:  PR[GP1:91,2] = PR[GP1:90,2] + -13.403;
   1:L PR[91] 10mm/sec CNT100;
   1:  PR[GP1:91,1] = PR[GP1:90,1] + -63.574;
   1:  PR[GP1:91,2] = PR[GP1:90,2] + -18.214;
   1:L PR[91] 10mm/sec CNT100;
   1:  PR[GP1:91,1] = PR[GP1:90,1] + -61.114;
   1:  PR[GP1:91,2] = PR[GP1:90,2] + -22.059;
   1:L PR[91] 10mm/sec CNT100;
   1:  PR[GP1:91,1] = PR[GP1:90,1] + -57.010;
   1:  PR[GP1:91,2] = PR[GP1:90,2] + -26.051;
   1:L PR[91] 10mm/sec CNT100;
   1:  PR[GP1:91,1] = PR[GP1:90,1] + -54.512;
   1:  PR[GP1:91,2] = PR[GP1:90,2] + -28.122;
   1:L PR[91] 10mm/sec CNT100;
   1:  PR[GP1:91,1] = PR[GP1:90,1] + -48.765;
   1:  PR[GP1:91,2] = PR[GP1:90,2] + -31.656;
   1:L PR[91] 10mm/sec CNT100;
   1:  PR[GP1:91,1] = PR[GP1:90,1] + -40.668;
   1:  PR[GP1:91,2] = PR[GP1:90,2] + -34.618;
   1:L PR[91] 10mm/sec CNT100;
   1:  PR[GP1:91,1] = PR[GP1:90,1] + -32.930;
   1:  PR[GP1:91,2] = PR[GP1:90,2] + -35.719;
   1:L PR[91] 10mm/sec CNT100;
   1:  PR[GP1:91,1] = PR[GP1:90,1] + -31.911;
   1:  PR[GP1:91,2] = PR[GP1:90,2] + -35.816;
   1:L PR[91] 10mm/sec CNT100;
   1:  PR[GP1:91,1] = PR[GP1:90,1] + -24.338;
   1:  PR[GP1:91,2] = PR[GP1:90,2] + -35.317;
   1:L PR[91] 10mm/sec CNT100;
   1:  PR[GP1:91,1] = PR[GP1:90,1] + -22.655;
   1:  PR[GP1:91,2] = PR[GP1:90,2] + -34.932;
   1:L PR[91] 10mm/sec CNT100;
   1:  PR[GP1:91,1] = PR[GP1:90,1] + -15.598;
   1:  PR[GP1:91,2] = PR[GP1:90,2] + -32.905;
   1:L PR[91] 10mm/sec CNT100;
   1:  PR[GP1:91,1] = PR[GP1:90,1] + -13.772;
   1:  PR[GP1:91,2] = PR[GP1:90,2] + -31.835;
   1:L PR[91] 10mm/sec CNT100;
   1:  PR[GP1:91,1] = PR[GP1:90,1] + -8.446;
   1:  PR[GP1:91,2] = PR[GP1:90,2] + -28.936;
   1:L PR[91] 10mm/sec CNT100;
   1:  PR[GP1:91,1] = PR[GP1:90,1] + -4.938;
   1:  PR[GP1:91,2] = PR[GP1:90,2] + -25.909;
   1:L PR[91] 10mm/sec CNT100;
   1:  PR[GP1:91,1] = PR[GP1:90,1] + -2.710;
   1:  PR[GP1:91,2] = PR[GP1:90,2] + -23.948;
   1:L PR[91] 10mm/sec CNT100;
   1:  PR[GP1:91,1] = PR[GP1:90,1] + -0.822;
   1:  PR[GP1:91,2] = PR[GP1:90,2] + -21.657;
   1:L PR[91] 10mm/sec CNT100;
   1:  PR[GP1:91,1] = PR[GP1:90,1] + 0.307;
   1:L PR[91] 10mm/sec CNT100;
   1:  PR[GP1:91,1] = PR[GP1:90,1] + 1.975;
   1:  PR[GP1:91,2] = PR[GP1:90,2] + -24.049;
   1:  PR[GP1:91,3] = PR[GP1:90,3] + 49.105;
   1:L PR[91] 10mm/sec CNT100;
   1:  PR[GP1:91,1] = PR[GP1:90,1] + 3.947;
   1:  PR[GP1:91,2] = PR[GP1:90,2] + -25.785;
   1:L PR[91] 10mm/sec CNT100;
   1:  PR[GP1:91,1] = PR[GP1:90,1] + 7.696;
   1:  PR[GP1:91,2] = PR[GP1:90,2] + -29.026;
   1:L PR[91] 10mm/sec CNT100;
   1:  PR[GP1:91,1] = PR[GP1:90,1] + 12.827;
   1:  PR[GP1:91,2] = PR[GP1:90,2] + -31.810;
   1:L PR[91] 10mm/sec CNT100;
   1:  PR[GP1:91,1] = PR[GP1:90,1] + 14.810;
   1:  PR[GP1:91,2] = PR[GP1:90,2] + -32.971;
   1:L PR[91] 10mm/sec CNT100;
   1:  PR[GP1:91,1] = PR[GP1:90,1] + 21.757;
   1:  PR[GP1:91,2] = PR[GP1:90,2] + -34.966;
   1:L PR[91] 10mm/sec CNT100;
   1:  PR[GP1:91,1] = PR[GP1:90,1] + 23.637;
   1:  PR[GP1:91,2] = PR[GP1:90,2] + -35.396;
   1:L PR[91] 10mm/sec CNT100;
   1:  PR[GP1:91,1] = PR[GP1:90,1] + 31.052;
   1:  PR[GP1:91,2] = PR[GP1:90,2] + -35.889;
   1:L PR[91] 10mm/sec CNT100;
   1:  PR[GP1:91,1] = PR[GP1:90,1] + 39.321;
   1:  PR[GP1:91,2] = PR[GP1:90,2] + -34.747;
   1:L PR[91] 10mm/sec CNT100;
   1:  PR[GP1:91,1] = PR[GP1:90,1] + 39.894;
   1:  PR[GP1:91,2] = PR[GP1:90,2] + -34.692;
   1:L PR[91] 10mm/sec CNT100;
   1:  PR[GP1:91,1] = PR[GP1:90,1] + 47.863;
   1:  PR[GP1:91,2] = PR[GP1:90,2] + -31.784;
   1:L PR[91] 10mm/sec CNT100;
   1:  PR[GP1:91,1] = PR[GP1:90,1] + 54.001;
   1:  PR[GP1:91,2] = PR[GP1:90,2] + -28.029;
   1:L PR[91] 10mm/sec CNT100;
   1:  PR[GP1:91,1] = PR[GP1:90,1] + 55.899;
   1:  PR[GP1:91,2] = PR[GP1:90,2] + -26.454;
   1:L PR[91] 10mm/sec CNT100;
   1:  PR[GP1:91,1] = PR[GP1:90,1] + 60.383;
   1:  PR[GP1:91,2] = PR[GP1:90,2] + -22.097;
   1:L PR[91] 10mm/sec CNT100;
   1:  PR[GP1:91,1] = PR[GP1:90,1] + 62.655;
   1:  PR[GP1:91,2] = PR[GP1:90,2] + -18.286;
   1:L PR[91] 10mm/sec CNT100;
   1:  PR[GP1:91,1] = PR[GP1:90,1] + 65.625;
   1:  PR[GP1:91,2] = PR[GP1:90,2] + -13.623;
   1:L PR[91] 10mm/sec CNT100;
   1:  PR[GP1:91,1] = PR[GP1:90,1] + 67.137;
   1:  PR[GP1:91,2] = PR[GP1:90,2] + -9.540;
   1:L PR[91] 10mm/sec CNT100;
   1:  PR[GP1:91,1] = PR[GP1:90,1] + 68.191;
   1:  PR[GP1:91,2] = PR[GP1:90,2] + -3.721;
   1:L PR[91] 10mm/sec CNT100;
   1:  PR[GP1:91,1] = PR[GP1:90,1] + 68.640;
   1:  PR[GP1:91,2] = PR[GP1:90,2] + 0.258;
   1:L PR[91] 10mm/sec CNT100;
   1:  PR[GP1:91,1] = PR[GP1:90,1] + 67.588;
   1:  PR[GP1:91,2] = PR[GP1:90,2] + 5.983;
   1:L PR[91] 10mm/sec CNT100;
   1:  PR[GP1:91,1] = PR[GP1:90,1] + 67.130;
   1:  PR[GP1:91,2] = PR[GP1:90,2] + 10.118;
   1:L PR[91] 10mm/sec CNT100;
   1:  PR[GP1:91,1] = PR[GP1:90,1] + 65.622;
   1:  PR[GP1:91,2] = PR[GP1:90,2] + 14.191;
   1:L PR[91] 10mm/sec CNT100;
   1:  PR[GP1:91,1] = PR[GP1:90,1] + 63.113;
   1:  PR[GP1:91,2] = PR[GP1:90,2] + 18.423;
   1:L PR[91] 10mm/sec CNT100;
   1:  PR[GP1:91,1] = PR[GP1:90,1] + 60.391;
   1:  PR[GP1:91,2] = PR[GP1:90,2] + 22.648;
   1:L PR[91] 10mm/sec CNT100;
   1:  PR[GP1:91,1] = PR[GP1:90,1] + 55.899;
   1:  PR[GP1:91,2] = PR[GP1:90,2] + 27.012;
   1:L PR[91] 10mm/sec CNT100;
   1:  PR[GP1:91,1] = PR[GP1:90,1] + 54.001;
   1:  PR[GP1:91,2] = PR[GP1:90,2] + 28.587;
   1:L PR[91] 10mm/sec CNT100;
   1:  PR[GP1:91,1] = PR[GP1:90,1] + 47.863;
   1:  PR[GP1:91,2] = PR[GP1:90,2] + 32.342;
   1:L PR[91] 10mm/sec CNT100;
   1:  PR[GP1:91,1] = PR[GP1:90,1] + 39.877;
   1:  PR[GP1:91,2] = PR[GP1:90,2] + 35.256;
   1:L PR[91] 10mm/sec CNT100;
   1:  PR[GP1:91,1] = PR[GP1:90,1] + 32.278;
   1:  PR[GP1:91,2] = PR[GP1:90,2] + 36.333;
   1:L PR[91] 10mm/sec CNT100;
   1:  PR[GP1:91,1] = PR[GP1:90,1] + 31.051;
   1:  PR[GP1:91,2] = PR[GP1:90,2] + 36.447;
   1:L PR[91] 10mm/sec CNT100;
   1:  PR[GP1:91,1] = PR[GP1:90,1] + 23.619;
   1:  PR[GP1:91,2] = PR[GP1:90,2] + 35.953;
   1:L PR[91] 10mm/sec CNT100;
   1:  PR[GP1:91,1] = PR[GP1:90,1] + 21.706;
   1:  PR[GP1:91,2] = PR[GP1:90,2] + 35.502;
   1:L PR[91] 10mm/sec CNT100;
   1:  PR[GP1:91,1] = PR[GP1:90,1] + 14.755;
   1:  PR[GP1:91,2] = PR[GP1:90,2] + 33.503;
   1:L PR[91] 10mm/sec CNT100;
   1:  PR[GP1:91,1] = PR[GP1:90,1] + 8.836;
   1:  PR[GP1:91,2] = PR[GP1:90,2] + 30.313;
   1:L PR[91] 10mm/sec CNT100;
   1:  PR[GP1:91,1] = PR[GP1:90,1] + 3.886;
   1:  PR[GP1:91,2] = PR[GP1:90,2] + 26.287;
   1:L PR[91] 10mm/sec CNT100;
   1:  PR[GP1:91,1] = PR[GP1:90,1] + 1.948;
   1:  PR[GP1:91,2] = PR[GP1:90,2] + 24.580;
   1:L PR[91] 10mm/sec CNT100;
   1:  PR[GP1:91,1] = PR[GP1:90,1] + 0.275;
   1:  PR[GP1:91,2] = PR[GP1:90,2] + 22.540;
   1:L PR[91] 10mm/sec CNT100;
   1:  PR[GP1:91,1] = PR[GP1:90,1] + -0.791;
   1:L PR[91] 10mm/sec CNT100;
   1:  PR[GP1:91,1] = PR[GP1:90,1] + -2.460;
   1:  PR[GP1:91,2] = PR[GP1:90,2] + 24.568;
   1:L PR[91] 10mm/sec CNT100;
   1:  PR[GP1:91,1] = PR[GP1:90,1] + -4.399;
   1:  PR[GP1:91,2] = PR[GP1:90,2] + 26.275;
   1:L PR[91] 10mm/sec CNT100;
   1:  PR[GP1:91,1] = PR[GP1:90,1] + -9.337;
   1:  PR[GP1:91,2] = PR[GP1:90,2] + 30.290;
   1:L PR[91] 10mm/sec CNT100;
   1:  PR[GP1:91,1] = PR[GP1:90,1] + -15.287;
   1:  PR[GP1:91,2] = PR[GP1:90,2] + 33.506;
   1:L PR[91] 10mm/sec CNT100;
   1:  PR[GP1:91,1] = PR[GP1:90,1] + -22.229;
   1:  PR[GP1:91,2] = PR[GP1:90,2] + 35.502;
   1:L PR[91] 10mm/sec CNT100;
   1:  PR[GP1:91,1] = PR[GP1:90,1] + -24.142;
   1:  PR[GP1:91,2] = PR[GP1:90,2] + 35.954;
   1:L PR[91] 10mm/sec CNT100;
   1:  PR[GP1:91,1] = PR[GP1:90,1] + -31.584;
   1:  PR[GP1:91,2] = PR[GP1:90,2] + 36.445;
   1:L PR[91] 10mm/sec CNT100;
   1:  PR[GP1:91,1] = PR[GP1:90,1] + -39.888;
   1:  PR[GP1:91,2] = PR[GP1:90,2] + 35.296;
   1:L PR[91] 10mm/sec CNT100;
   1:  PR[GP1:91,1] = PR[GP1:90,1] + -40.459;
   1:  PR[GP1:91,2] = PR[GP1:90,2] + 35.242;
   1:L PR[91] 10mm/sec CNT100;
   1:  PR[GP1:91,1] = PR[GP1:90,1] + -48.421;
   1:  PR[GP1:91,2] = PR[GP1:90,2] + 32.327;
   1:L PR[91] 10mm/sec CNT100;
   1:  PR[GP1:91,1] = PR[GP1:90,1] + -54.578;
   1:  PR[GP1:91,2] = PR[GP1:90,2] + 28.541;
   1:L PR[91] 10mm/sec CNT100;
   1:  PR[GP1:91,1] = PR[GP1:90,1] + -56.487;
   1:  PR[GP1:91,2] = PR[GP1:90,2] + 26.959;
   1:L PR[91] 10mm/sec CNT100;
   1:  PR[GP1:91,1] = PR[GP1:90,1] + -60.959;
   1:  PR[GP1:91,2] = PR[GP1:90,2] + 22.608;
   1:L PR[91] 10mm/sec CNT100;
   1:  PR[GP1:91,1] = PR[GP1:90,1] + -63.235;
   1:  PR[GP1:91,2] = PR[GP1:90,2] + 18.777;
   1:L PR[91] 10mm/sec CNT100;
   1:  PR[GP1:91,1] = PR[GP1:90,1] + -66.163;
   1:  PR[GP1:91,2] = PR[GP1:90,2] + 14.149;
   1:L PR[91] 10mm/sec CNT100;
   1:  PR[GP1:91,1] = PR[GP1:90,1] + -67.680;
   1:  PR[GP1:91,2] = PR[GP1:90,2] + 10.000;
   1:L PR[91] 10mm/sec CNT100;
   1:  PR[GP1:91,1] = PR[GP1:90,1] + -68.734;
   1:  PR[GP1:91,2] = PR[GP1:90,2] + 4.190;
   1:L PR[91] 10mm/sec CNT100;
   1:  PR[GP1:91,1] = PR[GP1:90,1] + -69.167;
   1:  PR[GP1:91,2] = PR[GP1:90,2] + 0.301;
   1:L PR[91] 10mm/sec CNT100;
   1:  PR[GP1:91,1] = PR[GP1:90,1] + -68.114;
   1:  PR[GP1:91,2] = PR[GP1:90,2] + -5.415;
   1:L PR[91] 10mm/sec CNT100;
   1:  PR[GP1:91,1] = PR[GP1:90,1] + -67.673;
   1:  PR[GP1:91,2] = PR[GP1:90,2] + -9.462;
   1:L PR[91] 10mm/sec CNT100;
   1:  PR[GP1:91,1] = PR[GP1:90,1] + -66.160;
   1:  PR[GP1:91,2] = PR[GP1:90,2] + -13.600;
   1:L PR[91] 10mm/sec CNT100;
   1:  PR[GP1:91,1] = PR[GP1:90,1] + -63.652;
   1:  PR[GP1:91,2] = PR[GP1:90,2] + -17.846;
   1:L PR[91] 10mm/sec CNT100;
   1:  PR[GP1:91,1] = PR[GP1:90,1] + -60.966;
   1:  PR[GP1:91,2] = PR[GP1:90,2] + -22.043;
   1:L PR[91] 10mm/sec CNT100;
   1:  PR[GP1:91,1] = PR[GP1:90,1] + -56.487;
   1:  PR[GP1:91,2] = PR[GP1:90,2] + -26.401;
   1:L PR[91] 10mm/sec CNT100;
   1:  PR[GP1:91,1] = PR[GP1:90,1] + -54.578;
   1:  PR[GP1:91,2] = PR[GP1:90,2] + -27.983;
   1:L PR[91] 10mm/sec CNT100;
   1:  PR[GP1:91,1] = PR[GP1:90,1] + -48.421;
   1:  PR[GP1:91,2] = PR[GP1:90,2] + -31.769;
   1:L PR[91] 10mm/sec CNT100;
   1:  PR[GP1:91,1] = PR[GP1:90,1] + -40.450;
   1:  PR[GP1:91,2] = PR[GP1:90,2] + -34.688;
   1:L PR[91] 10mm/sec CNT100;
   1:  PR[GP1:91,1] = PR[GP1:90,1] + -32.832;
   1:  PR[GP1:91,2] = PR[GP1:90,2] + -35.771;
   1:L PR[91] 10mm/sec CNT100;
   1:  PR[GP1:91,1] = PR[GP1:90,1] + -31.611;
   1:  PR[GP1:91,2] = PR[GP1:90,2] + -35.889;
   1:L PR[91] 10mm/sec CNT100;
   1:  PR[GP1:91,1] = PR[GP1:90,1] + -24.161;
   1:  PR[GP1:91,2] = PR[GP1:90,2] + -35.397;
   1:L PR[91] 10mm/sec CNT100;
   1:  PR[GP1:91,1] = PR[GP1:90,1] + -22.280;
   1:  PR[GP1:91,2] = PR[GP1:90,2] + -34.967;
   1:L PR[91] 10mm/sec CNT100;
   1:  PR[GP1:91,1] = PR[GP1:90,1] + -15.343;
   1:  PR[GP1:91,2] = PR[GP1:90,2] + -32.974;
   1:L PR[91] 10mm/sec CNT100;
   1:  PR[GP1:91,1] = PR[GP1:90,1] + -13.361;
   1:  PR[GP1:91,2] = PR[GP1:90,2] + -31.813;
   1:L PR[91] 10mm/sec CNT100;
   1:  PR[GP1:91,1] = PR[GP1:90,1] + -8.202;
   1:  PR[GP1:91,2] = PR[GP1:90,2] + -29.005;
   1:L PR[91] 10mm/sec CNT100;
   1:  PR[GP1:91,1] = PR[GP1:90,1] + -4.458;
   1:  PR[GP1:91,2] = PR[GP1:90,2] + -25.774;
   1:L PR[91] 10mm/sec CNT100;
   1:  PR[GP1:91,1] = PR[GP1:90,1] + -2.484;
   1:  PR[GP1:91,2] = PR[GP1:90,2] + -24.036;
   1:L PR[91] 10mm/sec CNT100;
   1:  PR[GP1:91,1] = PR[GP1:90,1] + -0.791;
   1:  PR[GP1:91,2] = PR[GP1:90,2] + -21.982;
   1:L PR[91] 10mm/sec CNT100;
   1:  PR[GP1:91,1] = PR[GP1:90,1] + 0.276;
   1:L PR[91] 10mm/sec CNT100;
   1:  PR[GP1:91,1] = PR[GP1:90,1] + 1.748;
   1:  PR[GP1:91,2] = PR[GP1:90,2] + -24.136;
   1:  PR[GP1:91,3] = PR[GP1:90,3] + 49.715;
   1:L PR[91] 10mm/sec CNT100;
   1:  PR[GP1:91,1] = PR[GP1:90,1] + 3.465;
   1:  PR[GP1:91,2] = PR[GP1:90,2] + -25.648;
   1:L PR[91] 10mm/sec CNT100;
   1:  PR[GP1:91,1] = PR[GP1:90,1] + 7.452;
   1:  PR[GP1:91,2] = PR[GP1:90,2] + -29.094;
   1:L PR[91] 10mm/sec CNT100;
   1:  PR[GP1:91,1] = PR[GP1:90,1] + 12.416;
   1:  PR[GP1:91,2] = PR[GP1:90,2] + -31.788;
   1:L PR[91] 10mm/sec CNT100;
   1:  PR[GP1:91,1] = PR[GP1:90,1] + 14.555;
   1:  PR[GP1:91,2] = PR[GP1:90,2] + -33.040;
   1:L PR[91] 10mm/sec CNT100;
   1:  PR[GP1:91,1] = PR[GP1:90,1] + 21.381;
   1:  PR[GP1:91,2] = PR[GP1:90,2] + -35.001;
   1:L PR[91] 10mm/sec CNT100;
   1:  PR[GP1:91,1] = PR[GP1:90,1] + 23.461;
   1:  PR[GP1:91,2] = PR[GP1:90,2] + -35.477;
   1:L PR[91] 10mm/sec CNT100;
   1:  PR[GP1:91,1] = PR[GP1:90,1] + 30.752;
   1:  PR[GP1:91,2] = PR[GP1:90,2] + -35.961;
   1:L PR[91] 10mm/sec CNT100;
   1:  PR[GP1:91,1] = PR[GP1:90,1] + 38.885;
   1:  PR[GP1:91,2] = PR[GP1:90,2] + -34.838;
   1:L PR[91] 10mm/sec CNT100;
   1:  PR[GP1:91,1] = PR[GP1:90,1] + 39.677;
   1:  PR[GP1:91,2] = PR[GP1:90,2] + -34.761;
   1:L PR[91] 10mm/sec CNT100;
   1:  PR[GP1:91,1] = PR[GP1:90,1] + 47.557;
   1:  PR[GP1:91,2] = PR[GP1:90,2] + -31.885;
   1:L PR[91] 10mm/sec CNT100;
   1:  PR[GP1:91,1] = PR[GP1:90,1] + 47.625;
   1:  PR[GP1:91,2] = PR[GP1:90,2] + -31.855;
   1:L PR[91] 10mm/sec CNT100;
   1:  PR[GP1:91,1] = PR[GP1:90,1] + 49.098;
   1:  PR[GP1:91,2] = PR[GP1:90,2] + -30.931;
   1:L PR[91] 10mm/sec CNT100;
   1:  PR[GP1:91,1] = PR[GP1:90,1] + 54.064;
   1:  PR[GP1:91,2] = PR[GP1:90,2] + -27.893;
   1:L PR[91] 10mm/sec CNT100;
   1:  PR[GP1:91,1] = PR[GP1:90,1] + 55.371;
   1:  PR[GP1:91,2] = PR[GP1:90,2] + -26.808;
   1:L PR[91] 10mm/sec CNT100;
   1:  PR[GP1:91,1] = PR[GP1:90,1] + 60.232;
   1:  PR[GP1:91,2] = PR[GP1:90,2] + -22.086;
   1:L PR[91] 10mm/sec CNT100;
   1:  PR[GP1:91,1] = PR[GP1:90,1] + 62.100;
   1:  PR[GP1:91,2] = PR[GP1:90,2] + -18.950;
   1:L PR[91] 10mm/sec CNT100;
   1:  PR[GP1:91,1] = PR[GP1:90,1] + 65.367;
   1:  PR[GP1:91,2] = PR[GP1:90,2] + -13.821;
   1:L PR[91] 10mm/sec CNT100;
   1:  PR[GP1:91,1] = PR[GP1:90,1] + 67.033;
   1:  PR[GP1:91,2] = PR[GP1:90,2] + -9.323;
   1:L PR[91] 10mm/sec CNT100;
   1:  PR[GP1:91,1] = PR[GP1:90,1] + 67.966;
   1:  PR[GP1:91,2] = PR[GP1:90,2] + -4.175;
   1:L PR[91] 10mm/sec CNT100;
   1:  PR[GP1:91,1] = PR[GP1:90,1] + 68.466;
   1:  PR[GP1:91,2] = PR[GP1:90,2] + 0.258;
   1:L PR[91] 10mm/sec CNT100;
   1:  PR[GP1:91,1] = PR[GP1:90,1] + 67.530;
   1:  PR[GP1:91,2] = PR[GP1:90,2] + 5.350;
   1:L PR[91] 10mm/sec CNT100;
   1:  PR[GP1:91,1] = PR[GP1:90,1] + 67.026;
   1:  PR[GP1:91,2] = PR[GP1:90,2] + 9.900;
   1:L PR[91] 10mm/sec CNT100;
   1:  PR[GP1:91,1] = PR[GP1:90,1] + 65.364;
   1:  PR[GP1:91,2] = PR[GP1:90,2] + 14.389;
   1:L PR[91] 10mm/sec CNT100;
   1:  PR[GP1:91,1] = PR[GP1:90,1] + 63.190;
   1:  PR[GP1:91,2] = PR[GP1:90,2] + 18.058;
   1:L PR[91] 10mm/sec CNT100;
   1:  PR[GP1:91,1] = PR[GP1:90,1] + 60.239;
   1:  PR[GP1:91,2] = PR[GP1:90,2] + 22.636;
   1:L PR[91] 10mm/sec CNT100;
   1:  PR[GP1:91,1] = PR[GP1:90,1] + 55.371;
   1:  PR[GP1:91,2] = PR[GP1:90,2] + 27.366;
   1:L PR[91] 10mm/sec CNT100;
   1:  PR[GP1:91,1] = PR[GP1:90,1] + 54.064;
   1:  PR[GP1:91,2] = PR[GP1:90,2] + 28.451;
   1:L PR[91] 10mm/sec CNT100;
   1:  PR[GP1:91,1] = PR[GP1:90,1] + 49.098;
   1:  PR[GP1:91,2] = PR[GP1:90,2] + 31.489;
   1:L PR[91] 10mm/sec CNT100;
   1:  PR[GP1:91,1] = PR[GP1:90,1] + 47.625;
   1:  PR[GP1:91,2] = PR[GP1:90,2] + 32.413;
   1:L PR[91] 10mm/sec CNT100;
   1:  PR[GP1:91,1] = PR[GP1:90,1] + 47.556;
   1:  PR[GP1:91,2] = PR[GP1:90,2] + 32.443;
   1:L PR[91] 10mm/sec CNT100;
   1:  PR[GP1:91,1] = PR[GP1:90,1] + 39.657;
   1:  PR[GP1:91,2] = PR[GP1:90,2] + 35.326;
   1:L PR[91] 10mm/sec CNT100;
   1:  PR[GP1:91,1] = PR[GP1:90,1] + 32.178;
   1:  PR[GP1:91,2] = PR[GP1:90,2] + 36.386;
   1:L PR[91] 10mm/sec CNT100;
   1:  PR[GP1:91,1] = PR[GP1:90,1] + 30.749;
   1:  PR[GP1:91,2] = PR[GP1:90,2] + 36.519;
   1:L PR[91] 10mm/sec CNT100;
   1:  PR[GP1:91,1] = PR[GP1:90,1] + 23.440;
   1:  PR[GP1:91,2] = PR[GP1:90,2] + 36.033;
   1:L PR[91] 10mm/sec CNT100;
   1:  PR[GP1:91,1] = PR[GP1:90,1] + 21.325;
   1:  PR[GP1:91,2] = PR[GP1:90,2] + 35.534;
   1:L PR[91] 10mm/sec CNT100;
   1:  PR[GP1:91,1] = PR[GP1:90,1] + 14.497;
   1:  PR[GP1:91,2] = PR[GP1:90,2] + 33.571;
   1:L PR[91] 10mm/sec CNT100;
   1:  PR[GP1:91,1] = PR[GP1:90,1] + 8.663;
   1:  PR[GP1:91,2] = PR[GP1:90,2] + 30.427;
   1:L PR[91] 10mm/sec CNT100;
   1:  PR[GP1:91,1] = PR[GP1:90,1] + 3.401;
   1:  PR[GP1:91,2] = PR[GP1:90,2] + 26.147;
   1:L PR[91] 10mm/sec CNT100;
   1:  PR[GP1:91,1] = PR[GP1:90,1] + 1.719;
   1:  PR[GP1:91,2] = PR[GP1:90,2] + 24.666;
   1:L PR[91] 10mm/sec CNT100;
   1:  PR[GP1:91,1] = PR[GP1:90,1] + 0.243;
   1:  PR[GP1:91,2] = PR[GP1:90,2] + 22.865;
   1:L PR[91] 10mm/sec CNT100;
   1:  PR[GP1:91,1] = PR[GP1:90,1] + -0.759;
   1:L PR[91] 10mm/sec CNT100;
   1:  PR[GP1:91,1] = PR[GP1:90,1] + -2.232;
   1:  PR[GP1:91,2] = PR[GP1:90,2] + 24.655;
   1:L PR[91] 10mm/sec CNT100;
   1:  PR[GP1:91,1] = PR[GP1:90,1] + -3.916;
   1:  PR[GP1:91,2] = PR[GP1:90,2] + 26.137;
   1:L PR[91] 10mm/sec CNT100;
   1:  PR[GP1:91,1] = PR[GP1:90,1] + -9.165;
   1:  PR[GP1:91,2] = PR[GP1:90,2] + 30.404;
   1:L PR[91] 10mm/sec CNT100;
   1:  PR[GP1:91,1] = PR[GP1:90,1] + -15.029;
   1:  PR[GP1:91,2] = PR[GP1:90,2] + 33.574;
   1:L PR[91] 10mm/sec CNT100;
   1:  PR[GP1:91,1] = PR[GP1:90,1] + -21.848;
   1:  PR[GP1:91,2] = PR[GP1:90,2] + 35.534;
   1:L PR[91] 10mm/sec CNT100;
   1:  PR[GP1:91,1] = PR[GP1:90,1] + -23.963;
   1:  PR[GP1:91,2] = PR[GP1:90,2] + 36.034;
   1:L PR[91] 10mm/sec CNT100;
   1:  PR[GP1:91,1] = PR[GP1:90,1] + -31.281;
   1:  PR[GP1:91,2] = PR[GP1:90,2] + 36.517;
   1:L PR[91] 10mm/sec CNT100;
   1:  PR[GP1:91,1] = PR[GP1:90,1] + -39.449;
   1:  PR[GP1:91,2] = PR[GP1:90,2] + 35.386;
   1:L PR[91] 10mm/sec CNT100;
   1:  PR[GP1:91,1] = PR[GP1:90,1] + -40.238;
   1:  PR[GP1:91,2] = PR[GP1:90,2] + 35.312;
   1:L PR[91] 10mm/sec CNT100;
   1:  PR[GP1:91,1] = PR[GP1:90,1] + -48.196;
   1:  PR[GP1:91,2] = PR[GP1:90,2] + 32.389;
   1:L PR[91] 10mm/sec CNT100;
   1:  PR[GP1:91,1] = PR[GP1:90,1] + -49.623;
   1:  PR[GP1:91,2] = PR[GP1:90,2] + 31.489;
   1:L PR[91] 10mm/sec CNT100;
   1:  PR[GP1:91,1] = PR[GP1:90,1] + -54.644;
   1:  PR[GP1:91,2] = PR[GP1:90,2] + 28.402;
   1:L PR[91] 10mm/sec CNT100;
   1:  PR[GP1:91,1] = PR[GP1:90,1] + -55.964;
   1:  PR[GP1:91,2] = PR[GP1:90,2] + 27.308;
   1:L PR[91] 10mm/sec CNT100;
   1:  PR[GP1:91,1] = PR[GP1:90,1] + -60.811;
   1:  PR[GP1:91,2] = PR[GP1:90,2] + 22.592;
   1:L PR[91] 10mm/sec CNT100;
   1:  PR[GP1:91,1] = PR[GP1:90,1] + -62.685;
   1:  PR[GP1:91,2] = PR[GP1:90,2] + 19.437;
   1:L PR[91] 10mm/sec CNT100;
   1:  PR[GP1:91,1] = PR[GP1:90,1] + -65.907;
   1:  PR[GP1:91,2] = PR[GP1:90,2] + 14.346;
   1:L PR[91] 10mm/sec CNT100;
   1:  PR[GP1:91,1] = PR[GP1:90,1] + -67.578;
   1:  PR[GP1:91,2] = PR[GP1:90,2] + 9.774;
   1:L PR[91] 10mm/sec CNT100;
   1:  PR[GP1:91,1] = PR[GP1:90,1] + -68.511;
   1:  PR[GP1:91,2] = PR[GP1:90,2] + 4.634;
   1:L PR[91] 10mm/sec CNT100;
   1:  PR[GP1:91,1] = PR[GP1:90,1] + -68.993;
   1:  PR[GP1:91,2] = PR[GP1:90,2] + 0.301;
   1:L PR[91] 10mm/sec CNT100;
   1:  PR[GP1:91,1] = PR[GP1:90,1] + -68.056;
   1:  PR[GP1:91,2] = PR[GP1:90,2] + -4.783;
   1:L PR[91] 10mm/sec CNT100;
   1:  PR[GP1:91,1] = PR[GP1:90,1] + -67.571;
   1:  PR[GP1:91,2] = PR[GP1:90,2] + -9.236;
   1:L PR[91] 10mm/sec CNT100;
   1:  PR[GP1:91,1] = PR[GP1:90,1] + -65.904;
   1:  PR[GP1:91,2] = PR[GP1:90,2] + -13.797;
   1:L PR[91] 10mm/sec CNT100;
   1:  PR[GP1:91,1] = PR[GP1:90,1] + -63.729;
   1:  PR[GP1:91,2] = PR[GP1:90,2] + -17.478;
   1:L PR[91] 10mm/sec CNT100;
   1:  PR[GP1:91,1] = PR[GP1:90,1] + -60.818;
   1:  PR[GP1:91,2] = PR[GP1:90,2] + -22.027;
   1:L PR[91] 10mm/sec CNT100;
   1:  PR[GP1:91,1] = PR[GP1:90,1] + -55.964;
   1:  PR[GP1:91,2] = PR[GP1:90,2] + -26.750;
   1:L PR[91] 10mm/sec CNT100;
   1:  PR[GP1:91,1] = PR[GP1:90,1] + -54.644;
   1:  PR[GP1:91,2] = PR[GP1:90,2] + -27.844;
   1:L PR[91] 10mm/sec CNT100;
   1:  PR[GP1:91,1] = PR[GP1:90,1] + -49.623;
   1:  PR[GP1:91,2] = PR[GP1:90,2] + -30.931;
   1:L PR[91] 10mm/sec CNT100;
   1:  PR[GP1:91,1] = PR[GP1:90,1] + -48.196;
   1:  PR[GP1:91,2] = PR[GP1:90,2] + -31.831;
   1:L PR[91] 10mm/sec CNT100;
   1:  PR[GP1:91,1] = PR[GP1:90,1] + -40.232;
   1:  PR[GP1:91,2] = PR[GP1:90,2] + -34.757;
   1:L PR[91] 10mm/sec CNT100;
   1:  PR[GP1:91,1] = PR[GP1:90,1] + -32.734;
   1:  PR[GP1:91,2] = PR[GP1:90,2] + -35.824;
   1:L PR[91] 10mm/sec CNT100;
   1:  PR[GP1:91,1] = PR[GP1:90,1] + -31.311;
   1:  PR[GP1:91,2] = PR[GP1:90,2] + -35.961;
   1:L PR[91] 10mm/sec CNT100;
   1:  PR[GP1:91,1] = PR[GP1:90,1] + -23.984;
   1:  PR[GP1:91,2] = PR[GP1:90,2] + -35.477;
   1:L PR[91] 10mm/sec CNT100;
   1:  PR[GP1:91,1] = PR[GP1:90,1] + -21.905;
   1:  PR[GP1:91,2] = PR[GP1:90,2] + -35.001;
   1:L PR[91] 10mm/sec CNT100;
   1:  PR[GP1:91,1] = PR[GP1:90,1] + -15.088;
   1:  PR[GP1:91,2] = PR[GP1:90,2] + -33.044;
   1:L PR[91] 10mm/sec CNT100;
   1:  PR[GP1:91,1] = PR[GP1:90,1] + -12.951;
   1:  PR[GP1:91,2] = PR[GP1:90,2] + -31.791;
   1:L PR[91] 10mm/sec CNT100;
   1:  PR[GP1:91,1] = PR[GP1:90,1] + -7.959;
   1:  PR[GP1:91,2] = PR[GP1:90,2] + -29.074;
   1:L PR[91] 10mm/sec CNT100;
   1:  PR[GP1:91,1] = PR[GP1:90,1] + -3.978;
   1:  PR[GP1:91,2] = PR[GP1:90,2] + -25.639;
   1:L PR[91] 10mm/sec CNT100;
   1:  PR[GP1:91,1] = PR[GP1:90,1] + -2.258;
   1:  PR[GP1:91,2] = PR[GP1:90,2] + -24.125;
   1:L PR[91] 10mm/sec CNT100;
   1:  PR[GP1:91,1] = PR[GP1:90,1] + -0.760;
   1:  PR[GP1:91,2] = PR[GP1:90,2] + -22.307;
   1:L PR[91] 10mm/sec CNT100;
   1:  PR[GP1:91,1] = PR[GP1:90,1] + 0.244;
   1:L PR[91] 10mm/sec CNT100;
   1:  PR[GP1:91,1] = PR[GP1:90,1] + 1.520;
   1:  PR[GP1:91,2] = PR[GP1:90,2] + -24.223;
   1:  PR[GP1:91,3] = PR[GP1:90,3] + 50.325;
   1:L PR[91] 10mm/sec CNT100;
   1:  PR[GP1:91,1] = PR[GP1:90,1] + 2.983;
   1:  PR[GP1:91,2] = PR[GP1:90,2] + -25.512;
   1:L PR[91] 10mm/sec CNT100;
   1:  PR[GP1:91,1] = PR[GP1:90,1] + 7.207;
   1:  PR[GP1:91,2] = PR[GP1:90,2] + -29.162;
   1:L PR[91] 10mm/sec CNT100;
   1:  PR[GP1:91,1] = PR[GP1:90,1] + 12.006;
   1:  PR[GP1:91,2] = PR[GP1:90,2] + -31.766;
   1:L PR[91] 10mm/sec CNT100;
   1:  PR[GP1:91,1] = PR[GP1:90,1] + 14.301;
   1:  PR[GP1:91,2] = PR[GP1:90,2] + -33.110;
   1:L PR[91] 10mm/sec CNT100;
   1:  PR[GP1:91,1] = PR[GP1:90,1] + 21.006;
   1:  PR[GP1:91,2] = PR[GP1:90,2] + -35.035;
   1:L PR[91] 10mm/sec CNT100;
   1:  PR[GP1:91,1] = PR[GP1:90,1] + 23.284;
   1:  PR[GP1:91,2] = PR[GP1:90,2] + -35.557;
   1:L PR[91] 10mm/sec CNT100;
   1:  PR[GP1:91,1] = PR[GP1:90,1] + 30.452;
   1:  PR[GP1:91,2] = PR[GP1:90,2] + -36.033;
   1:L PR[91] 10mm/sec CNT100;
   1:  PR[GP1:91,1] = PR[GP1:90,1] + 38.449;
   1:  PR[GP1:91,2] = PR[GP1:90,2] + -34.929;
   1:L PR[91] 10mm/sec CNT100;
   1:  PR[GP1:91,1] = PR[GP1:90,1] + 39.459;
   1:  PR[GP1:91,2] = PR[GP1:90,2] + -34.831;
   1:L PR[91] 10mm/sec CNT100;
   1:  PR[GP1:91,1] = PR[GP1:90,1] + 47.212;
   1:  PR[GP1:91,2] = PR[GP1:90,2] + -32.001;
   1:L PR[91] 10mm/sec CNT100;
   1:  PR[GP1:91,1] = PR[GP1:90,1] + 47.479;
   1:  PR[GP1:91,2] = PR[GP1:90,2] + -31.883;
   1:L PR[91] 10mm/sec CNT100;
   1:  PR[GP1:91,1] = PR[GP1:90,1] + 51.335;
   1:  PR[GP1:91,2] = PR[GP1:90,2] + -29.464;
   1:L PR[91] 10mm/sec CNT100;
   1:  PR[GP1:91,1] = PR[GP1:90,1] + 54.126;
   1:  PR[GP1:91,2] = PR[GP1:90,2] + -27.757;
   1:L PR[91] 10mm/sec CNT100;
   1:  PR[GP1:91,1] = PR[GP1:90,1] + 54.843;
   1:  PR[GP1:91,2] = PR[GP1:90,2] + -27.162;
   1:L PR[91] 10mm/sec CNT100;
   1:  PR[GP1:91,1] = PR[GP1:90,1] + 60.080;
   1:  PR[GP1:91,2] = PR[GP1:90,2] + -22.075;
   1:L PR[91] 10mm/sec CNT100;
   1:  PR[GP1:91,1] = PR[GP1:90,1] + 61.546;
   1:  PR[GP1:91,2] = PR[GP1:90,2] + -19.615;
   1:L PR[91] 10mm/sec CNT100;
   1:  PR[GP1:91,1] = PR[GP1:90,1] + 65.110;
   1:  PR[GP1:91,2] = PR[GP1:90,2] + -14.019;
   1:L PR[91] 10mm/sec CNT100;
   1:  PR[GP1:91,1] = PR[GP1:90,1] + 66.930;
   1:  PR[GP1:91,2] = PR[GP1:90,2] + -9.105;
   1:L PR[91] 10mm/sec CNT100;
   1:  PR[GP1:91,1] = PR[GP1:90,1] + 67.741;
   1:  PR[GP1:91,2] = PR[GP1:90,2] + -4.628;
   1:L PR[91] 10mm/sec CNT100;
   1:  PR[GP1:91,1] = PR[GP1:90,1] + 68.293;
   1:  PR[GP1:91,2] = PR[GP1:90,2] + 0.258;
   1:L PR[91] 10mm/sec CNT100;
   1:  PR[GP1:91,1] = PR[GP1:90,1] + 67.472;
   1:  PR[GP1:91,2] = PR[GP1:90,2] + 4.717;
   1:L PR[91] 10mm/sec CNT100;
   1:  PR[GP1:91,1] = PR[GP1:90,1] + 66.923;
   1:  PR[GP1:91,2] = PR[GP1:90,2] + 9.683;
   1:L PR[91] 10mm/sec CNT100;
   1:  PR[GP1:91,1] = PR[GP1:90,1] + 65.107;
   1:  PR[GP1:91,2] = PR[GP1:90,2] + 14.587;
   1:L PR[91] 10mm/sec CNT100;
   1:  PR[GP1:91,1] = PR[GP1:90,1] + 63.266;
   1:  PR[GP1:91,2] = PR[GP1:90,2] + 17.692;
   1:L PR[91] 10mm/sec CNT100;
   1:  PR[GP1:91,1] = PR[GP1:90,1] + 60.087;
   1:  PR[GP1:91,2] = PR[GP1:90,2] + 22.625;
   1:L PR[91] 10mm/sec CNT100;
   1:  PR[GP1:91,1] = PR[GP1:90,1] + 54.843;
   1:  PR[GP1:91,2] = PR[GP1:90,2] + 27.720;
   1:L PR[91] 10mm/sec CNT100;
   1:  PR[GP1:91,1] = PR[GP1:90,1] + 54.127;
   1:  PR[GP1:91,2] = PR[GP1:90,2] + 28.315;
   1:L PR[91] 10mm/sec CNT100;
   1:  PR[GP1:91,1] = PR[GP1:90,1] + 51.335;
   1:  PR[GP1:91,2] = PR[GP1:90,2] + 30.022;
   1:L PR[91] 10mm/sec CNT100;
   1:  PR[GP1:91,1] = PR[GP1:90,1] + 47.478;
   1:  PR[GP1:91,2] = PR[GP1:90,2] + 32.442;
   1:L PR[91] 10mm/sec CNT100;
   1:  PR[GP1:91,1] = PR[GP1:90,1] + 47.210;
   1:  PR[GP1:91,2] = PR[GP1:90,2] + 32.560;
   1:L PR[91] 10mm/sec CNT100;
   1:  PR[GP1:91,1] = PR[GP1:90,1] + 39.438;
   1:  PR[GP1:91,2] = PR[GP1:90,2] + 35.396;
   1:L PR[91] 10mm/sec CNT100;
   1:  PR[GP1:91,1] = PR[GP1:90,1] + 32.079;
   1:  PR[GP1:91,2] = PR[GP1:90,2] + 36.439;
   1:L PR[91] 10mm/sec CNT100;
   1:  PR[GP1:91,1] = PR[GP1:90,1] + 30.446;
   1:  PR[GP1:91,2] = PR[GP1:90,2] + 36.591;
   1:L PR[91] 10mm/sec CNT100;
   1:  PR[GP1:91,1] = PR[GP1:90,1] + 23.261;
   1:  PR[GP1:91,2] = PR[GP1:90,2] + 36.113;
   1:L PR[91] 10mm/sec CNT100;
   1:  PR[GP1:91,1] = PR[GP1:90,1] + 20.945;
   1:  PR[GP1:91,2] = PR[GP1:90,2] + 35.566;
   1:L PR[91] 10mm/sec CNT100;
   1:  PR[GP1:91,1] = PR[GP1:90,1] + 14.239;
   1:  PR[GP1:91,2] = PR[GP1:90,2] + 33.638;
   1:L PR[91] 10mm/sec CNT100;
   1:  PR[GP1:91,1] = PR[GP1:90,1] + 8.490;
   1:  PR[GP1:91,2] = PR[GP1:90,2] + 30.541;
   1:L PR[91] 10mm/sec CNT100;
   1:  PR[GP1:91,1] = PR[GP1:90,1] + 2.917;
   1:  PR[GP1:91,2] = PR[GP1:90,2] + 26.008;
   1:L PR[91] 10mm/sec CNT100;
   1:  PR[GP1:91,1] = PR[GP1:90,1] + 1.490;
   1:  PR[GP1:91,2] = PR[GP1:90,2] + 24.751;
   1:L PR[91] 10mm/sec CNT100;
   1:  PR[GP1:91,1] = PR[GP1:90,1] + 0.210;
   1:  PR[GP1:91,2] = PR[GP1:90,2] + 23.190;
   1:L PR[91] 10mm/sec CNT100;
   1:  PR[GP1:91,1] = PR[GP1:90,1] + -0.728;
   1:L PR[91] 10mm/sec CNT100;
   1:  PR[GP1:91,1] = PR[GP1:90,1] + -2.005;
   1:  PR[GP1:91,2] = PR[GP1:90,2] + 24.742;
   1:L PR[91] 10mm/sec CNT100;
   1:  PR[GP1:91,1] = PR[GP1:90,1] + -3.433;
   1:  PR[GP1:91,2] = PR[GP1:90,2] + 25.999;
   1:L PR[91] 10mm/sec CNT100;
   1:  PR[GP1:91,1] = PR[GP1:90,1] + -8.992;
   1:  PR[GP1:91,2] = PR[GP1:90,2] + 30.519;
   1:L PR[91] 10mm/sec CNT100;
   1:  PR[GP1:91,1] = PR[GP1:90,1] + -14.770;
   1:  PR[GP1:91,2] = PR[GP1:90,2] + 33.641;
   1:L PR[91] 10mm/sec CNT100;
   1:  PR[GP1:91,1] = PR[GP1:90,1] + -21.468;
   1:  PR[GP1:91,2] = PR[GP1:90,2] + 35.567;
   1:L PR[91] 10mm/sec CNT100;
   1:  PR[GP1:91,1] = PR[GP1:90,1] + -23.785;
   1:  PR[GP1:91,2] = PR[GP1:90,2] + 36.114;
   1:L PR[91] 10mm/sec CNT100;
   1:  PR[GP1:91,1] = PR[GP1:90,1] + -30.979;
   1:  PR[GP1:91,2] = PR[GP1:90,2] + 36.589;
   1:L PR[91] 10mm/sec CNT100;
   1:  PR[GP1:91,1] = PR[GP1:90,1] + -39.009;
   1:  PR[GP1:91,2] = PR[GP1:90,2] + 35.477;
   1:L PR[91] 10mm/sec CNT100;
   1:  PR[GP1:91,1] = PR[GP1:90,1] + -40.019;
   1:  PR[GP1:91,2] = PR[GP1:90,2] + 35.382;
   1:L PR[91] 10mm/sec CNT100;
   1:  PR[GP1:91,1] = PR[GP1:90,1] + -47.768;
   1:  PR[GP1:91,2] = PR[GP1:90,2] + 32.544;
   1:L PR[91] 10mm/sec CNT100;
   1:  PR[GP1:91,1] = PR[GP1:90,1] + -48.033;
   1:  PR[GP1:91,2] = PR[GP1:90,2] + 32.428;
   1:L PR[91] 10mm/sec CNT100;
   1:  PR[GP1:91,1] = PR[GP1:90,1] + -51.860;
   1:  PR[GP1:91,2] = PR[GP1:90,2] + 30.015;
   1:L PR[91] 10mm/sec CNT100;
   1:  PR[GP1:91,1] = PR[GP1:90,1] + -54.710;
   1:  PR[GP1:91,2] = PR[GP1:90,2] + 28.263;
   1:L PR[91] 10mm/sec CNT100;
   1:  PR[GP1:91,1] = PR[GP1:90,1] + -55.441;
   1:  PR[GP1:91,2] = PR[GP1:90,2] + 27.657;
   1:L PR[91] 10mm/sec CNT100;
   1:  PR[GP1:91,1] = PR[GP1:90,1] + -60.663;
   1:  PR[GP1:91,2] = PR[GP1:90,2] + 22.576;
   1:L PR[91] 10mm/sec CNT100;
   1:  PR[GP1:91,1] = PR[GP1:90,1] + -62.136;
   1:  PR[GP1:91,2] = PR[GP1:90,2] + 20.097;
   1:L PR[91] 10mm/sec CNT100;
   1:  PR[GP1:91,1] = PR[GP1:90,1] + -65.651;
   1:  PR[GP1:91,2] = PR[GP1:90,2] + 14.543;
   1:L PR[91] 10mm/sec CNT100;
   1:  PR[GP1:91,1] = PR[GP1:90,1] + -67.476;
   1:  PR[GP1:91,2] = PR[GP1:90,2] + 9.549;
   1:L PR[91] 10mm/sec CNT100;
   1:  PR[GP1:91,1] = PR[GP1:90,1] + -68.287;
   1:  PR[GP1:91,2] = PR[GP1:90,2] + 5.077;
   1:L PR[91] 10mm/sec CNT100;
   1:  PR[GP1:91,1] = PR[GP1:90,1] + -68.819;
   1:  PR[GP1:91,2] = PR[GP1:90,2] + 0.301;
   1:L PR[91] 10mm/sec CNT100;
   1:  PR[GP1:91,1] = PR[GP1:90,1] + -67.999;
   1:  PR[GP1:91,2] = PR[GP1:90,2] + -4.152;
   1:L PR[91] 10mm/sec CNT100;
   1:  PR[GP1:91,1] = PR[GP1:90,1] + -67.469;
   1:  PR[GP1:91,2] = PR[GP1:90,2] + -9.011;
   1:L PR[91] 10mm/sec CNT100;
   1:  PR[GP1:91,1] = PR[GP1:90,1] + -65.648;
   1:  PR[GP1:91,2] = PR[GP1:90,2] + -13.993;
   1:L PR[91] 10mm/sec CNT100;
   1:  PR[GP1:91,1] = PR[GP1:90,1] + -63.806;
   1:  PR[GP1:91,2] = PR[GP1:90,2] + -17.110;
   1:L PR[91] 10mm/sec CNT100;
   1:  PR[GP1:91,1] = PR[GP1:90,1] + -60.670;
   1:  PR[GP1:91,2] = PR[GP1:90,2] + -22.011;
   1:L PR[91] 10mm/sec CNT100;
   1:  PR[GP1:91,1] = PR[GP1:90,1] + -55.441;
   1:  PR[GP1:91,2] = PR[GP1:90,2] + -27.099;
   1:L PR[91] 10mm/sec CNT100;
   1:  PR[GP1:91,1] = PR[GP1:90,1] + -54.710;
   1:  PR[GP1:91,2] = PR[GP1:90,2] + -27.705;
   1:L PR[91] 10mm/sec CNT100;
   1:  PR[GP1:91,1] = PR[GP1:90,1] + -51.860;
   1:  PR[GP1:91,2] = PR[GP1:90,2] + -29.457;
   1:L PR[91] 10mm/sec CNT100;
   1:  PR[GP1:91,1] = PR[GP1:90,1] + -48.035;
   1:  PR[GP1:91,2] = PR[GP1:90,2] + -31.869;
   1:L PR[91] 10mm/sec CNT100;
   1:  PR[GP1:91,1] = PR[GP1:90,1] + -47.770;
   1:  PR[GP1:91,2] = PR[GP1:90,2] + -31.986;
   1:L PR[91] 10mm/sec CNT100;
   1:  PR[GP1:91,1] = PR[GP1:90,1] + -40.014;
   1:  PR[GP1:91,2] = PR[GP1:90,2] + -34.827;
   1:L PR[91] 10mm/sec CNT100;
   1:  PR[GP1:91,1] = PR[GP1:90,1] + -32.636;
   1:  PR[GP1:91,2] = PR[GP1:90,2] + -35.877;
   1:L PR[91] 10mm/sec CNT100;
   1:  PR[GP1:91,1] = PR[GP1:90,1] + -31.010;
   1:  PR[GP1:91,2] = PR[GP1:90,2] + -36.033;
   1:L PR[91] 10mm/sec CNT100;
   1:  PR[GP1:91,1] = PR[GP1:90,1] + -23.808;
   1:  PR[GP1:91,2] = PR[GP1:90,2] + -35.557;
   1:L PR[91] 10mm/sec CNT100;
   1:  PR[GP1:91,1] = PR[GP1:90,1] + -21.529;
   1:  PR[GP1:91,2] = PR[GP1:90,2] + -35.036;
   1:L PR[91] 10mm/sec CNT100;
   1:  PR[GP1:91,1] = PR[GP1:90,1] + -14.833;
   1:  PR[GP1:91,2] = PR[GP1:90,2] + -33.113;
   1:L PR[91] 10mm/sec CNT100;
   1:  PR[GP1:91,1] = PR[GP1:90,1] + -12.540;
   1:  PR[GP1:91,2] = PR[GP1:90,2] + -31.769;
   1:L PR[91] 10mm/sec CNT100;
   1:  PR[GP1:91,1] = PR[GP1:90,1] + -7.715;
   1:  PR[GP1:91,2] = PR[GP1:90,2] + -29.143;
   1:L PR[91] 10mm/sec CNT100;
   1:  PR[GP1:91,1] = PR[GP1:90,1] + -3.497;
   1:  PR[GP1:91,2] = PR[GP1:90,2] + -25.503;
   1:L PR[91] 10mm/sec CNT100;
   1:  PR[GP1:91,1] = PR[GP1:90,1] + -2.032;
   1:  PR[GP1:91,2] = PR[GP1:90,2] + -24.213;
   1:L PR[91] 10mm/sec CNT100;
   1:  PR[GP1:91,1] = PR[GP1:90,1] + -0.729;
   1:  PR[GP1:91,2] = PR[GP1:90,2] + -22.632;
   1:L PR[91] 10mm/sec CNT100;
   1:  PR[GP1:91,1] = PR[GP1:90,1] + 0.212;
   1:L PR[91] 10mm/sec CNT100;
   1:  PR[GP1:91,1] = PR[GP1:90,1] + 1.292;
   1:  PR[GP1:91,2] = PR[GP1:90,2] + -24.310;
   1:  PR[GP1:91,3] = PR[GP1:90,3] + 50.935;
   1:L PR[91] 10mm/sec CNT100;
   1:  PR[GP1:91,1] = PR[GP1:90,1] + 2.502;
   1:  PR[GP1:91,2] = PR[GP1:90,2] + -25.375;
   1:L PR[91] 10mm/sec CNT100;
   1:  PR[GP1:91,1] = PR[GP1:90,1] + 6.963;
   1:  PR[GP1:91,2] = PR[GP1:90,2] + -29.231;
   1:L PR[91] 10mm/sec CNT100;
   1:  PR[GP1:91,1] = PR[GP1:90,1] + 11.595;
   1:  PR[GP1:91,2] = PR[GP1:90,2] + -31.745;
   1:L PR[91] 10mm/sec CNT100;
   1:  PR[GP1:91,1] = PR[GP1:90,1] + 14.046;
   1:  PR[GP1:91,2] = PR[GP1:90,2] + -33.179;
   1:L PR[91] 10mm/sec CNT100;
   1:  PR[GP1:91,1] = PR[GP1:90,1] + 20.630;
   1:  PR[GP1:91,2] = PR[GP1:90,2] + -35.070;
   1:L PR[91] 10mm/sec CNT100;
   1:  PR[GP1:91,1] = PR[GP1:90,1] + 23.107;
   1:  PR[GP1:91,2] = PR[GP1:90,2] + -35.637;
   1:L PR[91] 10mm/sec CNT100;
   1:  PR[GP1:91,1] = PR[GP1:90,1] + 30.152;
   1:  PR[GP1:91,2] = PR[GP1:90,2] + -36.105;
   1:L PR[91] 10mm/sec CNT100;
   1:  PR[GP1:91,1] = PR[GP1:90,1] + 38.013;
   1:  PR[GP1:91,2] = PR[GP1:90,2] + -35.020;
   1:L PR[91] 10mm/sec CNT100;
   1:  PR[GP1:91,1] = PR[GP1:90,1] + 39.242;
   1:  PR[GP1:91,2] = PR[GP1:90,2] + -34.900;
   1:L PR[91] 10mm/sec CNT100;
   1:  PR[GP1:91,1] = PR[GP1:90,1] + 46.868;
   1:  PR[GP1:91,2] = PR[GP1:90,2] + -32.117;
   1:L PR[91] 10mm/sec CNT100;
   1:  PR[GP1:91,1] = PR[GP1:90,1] + 47.335;
   1:  PR[GP1:91,2] = PR[GP1:90,2] + -31.912;
   1:L PR[91] 10mm/sec CNT100;
   1:  PR[GP1:91,1] = PR[GP1:90,1] + 54.187;
   1:  PR[GP1:91,2] = PR[GP1:90,2] + -27.622;
   1:L PR[91] 10mm/sec CNT100;
   1:  PR[GP1:91,1] = PR[GP1:90,1] + 54.315;
   1:  PR[GP1:91,2] = PR[GP1:90,2] + -27.516;
   1:L PR[91] 10mm/sec CNT100;
   1:  PR[GP1:91,1] = PR[GP1:90,1] + 59.928;
   1:  PR[GP1:91,2] = PR[GP1:90,2] + -22.063;
   1:L PR[91] 10mm/sec CNT100;
   1:  PR[GP1:91,1] = PR[GP1:90,1] + 60.991;
   1:  PR[GP1:91,2] = PR[GP1:90,2] + -20.280;
   1:L PR[91] 10mm/sec CNT100;
   1:  PR[GP1:91,1] = PR[GP1:90,1] + 64.853;
   1:  PR[GP1:91,2] = PR[GP1:90,2] + -14.217;
   1:L PR[91] 10mm/sec CNT100;
   1:  PR[GP1:91,1] = PR[GP1:90,1] + 66.826;
   1:  PR[GP1:91,2] = PR[GP1:90,2] + -8.888;
   1:L PR[91] 10mm/sec CNT100;
   1:  PR[GP1:91,1] = PR[GP1:90,1] + 67.516;
   1:  PR[GP1:91,2] = PR[GP1:90,2] + -5.082;
   1:L PR[91] 10mm/sec CNT100;
   1:  PR[GP1:91,1] = PR[GP1:90,1] + 68.119;
   1:  PR[GP1:91,2] = PR[GP1:90,2] + 0.258;
   1:L PR[91] 10mm/sec CNT100;
   1:  PR[GP1:91,1] = PR[GP1:90,1] + 67.415;
   1:  PR[GP1:91,2] = PR[GP1:90,2] + 4.085;
   1:L PR[91] 10mm/sec CNT100;
   1:  PR[GP1:91,1] = PR[GP1:90,1] + 66.819;
   1:  PR[GP1:91,2] = PR[GP1:90,2] + 9.465;
   1:L PR[91] 10mm/sec CNT100;
   1:  PR[GP1:91,1] = PR[GP1:90,1] + 64.849;
   1:  PR[GP1:91,2] = PR[GP1:90,2] + 14.785;
   1:L PR[91] 10mm/sec CNT100;
   1:  PR[GP1:91,1] = PR[GP1:90,1] + 63.343;
   1:  PR[GP1:91,2] = PR[GP1:90,2] + 17.327;
   1:L PR[91] 10mm/sec CNT100;
   1:  PR[GP1:91,1] = PR[GP1:90,1] + 59.936;
   1:  PR[GP1:91,2] = PR[GP1:90,2] + 22.614;
   1:L PR[91] 10mm/sec CNT100;
   1:  PR[GP1:91,1] = PR[GP1:90,1] + 54.315;
   1:  PR[GP1:91,2] = PR[GP1:90,2] + 28.074;
   1:L PR[91] 10mm/sec CNT100;
   1:  PR[GP1:91,1] = PR[GP1:90,1] + 54.187;
   1:  PR[GP1:91,2] = PR[GP1:90,2] + 28.180;
   1:L PR[91] 10mm/sec CNT100;
   1:  PR[GP1:91,1] = PR[GP1:90,1] + 47.332;
   1:  PR[GP1:91,2] = PR[GP1:90,2] + 32.471;
   1:L PR[91] 10mm/sec CNT100;
   1:  PR[GP1:91,1] = PR[GP1:90,1] + 46.864;
   1:  PR[GP1:91,2] = PR[GP1:90,2] + 32.676;
   1:L PR[91] 10mm/sec CNT100;
   1:  PR[GP1:91,1] = PR[GP1:90,1] + 39.219;
   1:  PR[GP1:91,2] = PR[GP1:90,2] + 35.466;
   1:L PR[91] 10mm/sec CNT100;
   1:  PR[GP1:91,1] = PR[GP1:90,1] + 31.980;
   1:  PR[GP1:91,2] = PR[GP1:90,2] + 36.492;
   1:L PR[91] 10mm/sec CNT100;
   1:  PR[GP1:91,1] = PR[GP1:90,1] + 30.144;
   1:  PR[GP1:91,2] = PR[GP1:90,2] + 36.663;
   1:L PR[91] 10mm/sec CNT100;
   1:  PR[GP1:91,1] = PR[GP1:90,1] + 23.082;
   1:  PR[GP1:91,2] = PR[GP1:90,2] + 36.193;
   1:L PR[91] 10mm/sec CNT100;
   1:  PR[GP1:91,1] = PR[GP1:90,1] + 20.564;
   1:  PR[GP1:91,2] = PR[GP1:90,2] + 35.599;
   1:L PR[91] 10mm/sec CNT100;
   1:  PR[GP1:91,1] = PR[GP1:90,1] + 13.980;
   1:  PR[GP1:91,2] = PR[GP1:90,2] + 33.706;
   1:L PR[91] 10mm/sec CNT100;
   1:  PR[GP1:91,1] = PR[GP1:90,1] + 8.317;
   1:  PR[GP1:91,2] = PR[GP1:90,2] + 30.655;
   1:L PR[91] 10mm/sec CNT100;
   1:  PR[GP1:91,1] = PR[GP1:90,1] + 2.432;
   1:  PR[GP1:91,2] = PR[GP1:90,2] + 25.868;
   1:L PR[91] 10mm/sec CNT100;
   1:  PR[GP1:91,1] = PR[GP1:90,1] + 1.261;
   1:  PR[GP1:91,2] = PR[GP1:90,2] + 24.837;
   1:L PR[91] 10mm/sec CNT100;
   1:  PR[GP1:91,1] = PR[GP1:90,1] + 0.177;
   1:  PR[GP1:91,2] = PR[GP1:90,2] + 23.515;
   1:L PR[91] 10mm/sec CNT100;
   1:  PR[GP1:91,1] = PR[GP1:90,1] + -0.696;
   1:L PR[91] 10mm/sec CNT100;
   1:  PR[GP1:91,1] = PR[GP1:90,1] + -1.778;
   1:  PR[GP1:91,2] = PR[GP1:90,2] + 24.829;
   1:L PR[91] 10mm/sec CNT100;
   1:  PR[GP1:91,1] = PR[GP1:90,1] + -2.950;
   1:  PR[GP1:91,2] = PR[GP1:90,2] + 25.861;
   1:L PR[91] 10mm/sec CNT100;
   1:  PR[GP1:91,1] = PR[GP1:90,1] + -8.820;
   1:  PR[GP1:91,2] = PR[GP1:90,2] + 30.633;
   1:L PR[91] 10mm/sec CNT100;
   1:  PR[GP1:91,1] = PR[GP1:90,1] + -14.512;
   1:  PR[GP1:91,2] = PR[GP1:90,2] + 33.709;
   1:L PR[91] 10mm/sec CNT100;
   1:  PR[GP1:91,1] = PR[GP1:90,1] + -21.087;
   1:  PR[GP1:91,2] = PR[GP1:90,2] + 35.599;
   1:L PR[91] 10mm/sec CNT100;
   1:  PR[GP1:91,1] = PR[GP1:90,1] + -23.606;
   1:  PR[GP1:91,2] = PR[GP1:90,2] + 36.194;
   1:L PR[91] 10mm/sec CNT100;
   1:  PR[GP1:91,1] = PR[GP1:90,1] + -30.676;
   1:  PR[GP1:91,2] = PR[GP1:90,2] + 36.660;
   1:L PR[91] 10mm/sec CNT100;
   1:  PR[GP1:91,1] = PR[GP1:90,1] + -38.570;
   1:  PR[GP1:91,2] = PR[GP1:90,2] + 35.568;
   1:L PR[91] 10mm/sec CNT100;
   1:  PR[GP1:91,1] = PR[GP1:90,1] + -39.799;
   1:  PR[GP1:91,2] = PR[GP1:90,2] + 35.452;
   1:L PR[91] 10mm/sec CNT100;
   1:  PR[GP1:91,1] = PR[GP1:90,1] + -47.421;
   1:  PR[GP1:91,2] = PR[GP1:90,2] + 32.661;
   1:L PR[91] 10mm/sec CNT100;
   1:  PR[GP1:91,1] = PR[GP1:90,1] + -47.887;
   1:  PR[GP1:91,2] = PR[GP1:90,2] + 32.457;
   1:L PR[91] 10mm/sec CNT100;
   1:  PR[GP1:91,1] = PR[GP1:90,1] + -54.774;
   1:  PR[GP1:91,2] = PR[GP1:90,2] + 28.126;
   1:L PR[91] 10mm/sec CNT100;
   1:  PR[GP1:91,1] = PR[GP1:90,1] + -54.918;
   1:  PR[GP1:91,2] = PR[GP1:90,2] + 28.006;
   1:L PR[91] 10mm/sec CNT100;
   1:  PR[GP1:91,1] = PR[GP1:90,1] + -60.515;
   1:  PR[GP1:91,2] = PR[GP1:90,2] + 22.560;
   1:L PR[91] 10mm/sec CNT100;
   1:  PR[GP1:91,1] = PR[GP1:90,1] + -61.586;
   1:  PR[GP1:91,2] = PR[GP1:90,2] + 20.757;
   1:L PR[91] 10mm/sec CNT100;
   1:  PR[GP1:91,1] = PR[GP1:90,1] + -65.395;
   1:  PR[GP1:91,2] = PR[GP1:90,2] + 14.740;
   1:L PR[91] 10mm/sec CNT100;
   1:  PR[GP1:91,1] = PR[GP1:90,1] + -67.374;
   1:  PR[GP1:91,2] = PR[GP1:90,2] + 9.324;
   1:L PR[91] 10mm/sec CNT100;
   1:  PR[GP1:91,1] = PR[GP1:90,1] + -68.064;
   1:  PR[GP1:91,2] = PR[GP1:90,2] + 5.521;
   1:L PR[91] 10mm/sec CNT100;
   1:  PR[GP1:91,1] = PR[GP1:90,1] + -68.645;
   1:  PR[GP1:91,2] = PR[GP1:90,2] + 0.301;
   1:L PR[91] 10mm/sec CNT100;
   1:  PR[GP1:91,1] = PR[GP1:90,1] + -67.941;
   1:  PR[GP1:91,2] = PR[GP1:90,2] + -3.520;
   1:L PR[91] 10mm/sec CNT100;
   1:  PR[GP1:91,1] = PR[GP1:90,1] + -67.367;
   1:  PR[GP1:91,2] = PR[GP1:90,2] + -8.786;
   1:L PR[91] 10mm/sec CNT100;
   1:  PR[GP1:91,1] = PR[GP1:90,1] + -65.392;
   1:  PR[GP1:91,2] = PR[GP1:90,2] + -14.190;
   1:L PR[91] 10mm/sec CNT100;
   1:  PR[GP1:91,1] = PR[GP1:90,1] + -63.884;
   1:  PR[GP1:91,2] = PR[GP1:90,2] + -16.743;
   1:L PR[91] 10mm/sec CNT100;
   1:  PR[GP1:91,1] = PR[GP1:90,1] + -60.522;
   1:  PR[GP1:91,2] = PR[GP1:90,2] + -21.995;
   1:L PR[91] 10mm/sec CNT100;
   1:  PR[GP1:91,1] = PR[GP1:90,1] + -54.918;
   1:  PR[GP1:91,2] = PR[GP1:90,2] + -27.448;
   1:L PR[91] 10mm/sec CNT100;
   1:  PR[GP1:91,1] = PR[GP1:90,1] + -54.774;
   1:  PR[GP1:91,2] = PR[GP1:90,2] + -27.568;
   1:L PR[91] 10mm/sec CNT100;
   1:  PR[GP1:91,1] = PR[GP1:90,1] + -47.889;
   1:  PR[GP1:91,2] = PR[GP1:90,2] + -31.898;
   1:L PR[91] 10mm/sec CNT100;
   1:  PR[GP1:91,1] = PR[GP1:90,1] + -47.426;
   1:  PR[GP1:91,2] = PR[GP1:90,2] + -32.102;
   1:L PR[91] 10mm/sec CNT100;
   1:  PR[GP1:91,1] = PR[GP1:90,1] + -39.796;
   1:  PR[GP1:91,2] = PR[GP1:90,2] + -34.897;
   1:L PR[91] 10mm/sec CNT100;
   1:  PR[GP1:91,1] = PR[GP1:90,1] + -32.538;
   1:  PR[GP1:91,2] = PR[GP1:90,2] + -35.929;
   1:L PR[91] 10mm/sec CNT100;
   1:  PR[GP1:91,1] = PR[GP1:90,1] + -30.710;
   1:  PR[GP1:91,2] = PR[GP1:90,2] + -36.105;
   1:L PR[91] 10mm/sec CNT100;
   1:  PR[GP1:91,1] = PR[GP1:90,1] + -23.631;
   1:  PR[GP1:91,2] = PR[GP1:90,2] + -35.637;
   1:L PR[91] 10mm/sec CNT100;
   1:  PR[GP1:91,1] = PR[GP1:90,1] + -21.154;
   1:  PR[GP1:91,2] = PR[GP1:90,2] + -35.071;
   1:L PR[91] 10mm/sec CNT100;
   1:  PR[GP1:91,1] = PR[GP1:90,1] + -14.579;
   1:  PR[GP1:91,2] = PR[GP1:90,2] + -33.182;
   1:L PR[91] 10mm/sec CNT100;
   1:  PR[GP1:91,1] = PR[GP1:90,1] + -12.129;
   1:  PR[GP1:91,2] = PR[GP1:90,2] + -31.748;
   1:L PR[91] 10mm/sec CNT100;
   1:  PR[GP1:91,1] = PR[GP1:90,1] + -7.472;
   1:  PR[GP1:91,2] = PR[GP1:90,2] + -29.212;
   1:L PR[91] 10mm/sec CNT100;
   1:  PR[GP1:91,1] = PR[GP1:90,1] + -3.018;
   1:  PR[GP1:91,2] = PR[GP1:90,2] + -25.369;
   1:L PR[91] 10mm/sec CNT100;
   1:  PR[GP1:91,1] = PR[GP1:90,1] + -1.806;
   1:  PR[GP1:91,2] = PR[GP1:90,2] + -24.302;
   1:L PR[91] 10mm/sec CNT100;
   1:  PR[GP1:91,1] = PR[GP1:90,1] + -0.697;
   1:  PR[GP1:91,2] = PR[GP1:90,2] + -22.957;
   1:L PR[91] 10mm/sec CNT100;
   1:  PR[GP1:91,1] = PR[GP1:90,1] + 0.180;
   1:L PR[91] 10mm/sec CNT100;
   1:  PR[GP1:91,1] = PR[GP1:90,1] + 1.065;
   1:  PR[GP1:91,2] = PR[GP1:90,2] + -24.397;
   1:  PR[GP1:91,3] = PR[GP1:90,3] + 51.545;
   1:L PR[91] 10mm/sec CNT100;
   1:  PR[GP1:91,1] = PR[GP1:90,1] + 2.021;
   1:  PR[GP1:91,2] = PR[GP1:90,2] + -25.239;
   1:L PR[91] 10mm/sec CNT100;
   1:  PR[GP1:91,1] = PR[GP1:90,1] + 6.718;
   1:  PR[GP1:91,2] = PR[GP1:90,2] + -29.299;
   1:L PR[91] 10mm/sec CNT100;
   1:  PR[GP1:91,1] = PR[GP1:90,1] + 11.184;
   1:  PR[GP1:91,2] = PR[GP1:90,2] + -31.723;
   1:L PR[91] 10mm/sec CNT100;
   1:  PR[GP1:91,1] = PR[GP1:90,1] + 13.791;
   1:  PR[GP1:91,2] = PR[GP1:90,2] + -33.249;
   1:L PR[91] 10mm/sec CNT100;
   1:  PR[GP1:91,1] = PR[GP1:90,1] + 20.255;
   1:  PR[GP1:91,2] = PR[GP1:90,2] + -35.105;
   1:L PR[91] 10mm/sec CNT100;
   1:  PR[GP1:91,1] = PR[GP1:90,1] + 22.930;
   1:  PR[GP1:91,2] = PR[GP1:90,2] + -35.717;
   1:L PR[91] 10mm/sec CNT100;
   1:  PR[GP1:91,1] = PR[GP1:90,1] + 29.852;
   1:  PR[GP1:91,2] = PR[GP1:90,2] + -36.177;
   1:L PR[91] 10mm/sec CNT100;
   1:  PR[GP1:91,1] = PR[GP1:90,1] + 37.577;
   1:  PR[GP1:91,2] = PR[GP1:90,2] + -35.111;
   1:L PR[91] 10mm/sec CNT100;
   1:  PR[GP1:91,1] = PR[GP1:90,1] + 39.024;
   1:  PR[GP1:91,2] = PR[GP1:90,2] + -34.970;
   1:L PR[91] 10mm/sec CNT100;
   1:  PR[GP1:91,1] = PR[GP1:90,1] + 46.524;
   1:  PR[GP1:91,2] = PR[GP1:90,2] + -32.232;
   1:L PR[91] 10mm/sec CNT100;
   1:  PR[GP1:91,1] = PR[GP1:90,1] + 47.189;
   1:  PR[GP1:91,2] = PR[GP1:90,2] + -31.940;
   1:L PR[91] 10mm/sec CNT100;
   1:  PR[GP1:91,1] = PR[GP1:90,1] + 54.006;
   1:  PR[GP1:91,2] = PR[GP1:90,2] + -27.663;
   1:L PR[91] 10mm/sec CNT100;
   1:  PR[GP1:91,1] = PR[GP1:90,1] + 59.776;
   1:  PR[GP1:91,2] = PR[GP1:90,2] + -22.052;
   1:L PR[91] 10mm/sec CNT100;
   1:  PR[GP1:91,1] = PR[GP1:90,1] + 60.436;
   1:  PR[GP1:91,2] = PR[GP1:90,2] + -20.945;
   1:L PR[91] 10mm/sec CNT100;
   1:  PR[GP1:91,1] = PR[GP1:90,1] + 64.595;
   1:  PR[GP1:91,2] = PR[GP1:90,2] + -14.415;
   1:L PR[91] 10mm/sec CNT100;
   1:  PR[GP1:91,1] = PR[GP1:90,1] + 66.723;
   1:  PR[GP1:91,2] = PR[GP1:90,2] + -8.670;
   1:L PR[91] 10mm/sec CNT100;
   1:  PR[GP1:91,1] = PR[GP1:90,1] + 67.291;
   1:  PR[GP1:91,2] = PR[GP1:90,2] + -5.536;
   1:L PR[91] 10mm/sec CNT100;
   1:  PR[GP1:91,1] = PR[GP1:90,1] + 67.945;
   1:  PR[GP1:91,2] = PR[GP1:90,2] + 0.258;
   1:L PR[91] 10mm/sec CNT100;
   1:  PR[GP1:91,1] = PR[GP1:90,1] + 67.357;
   1:  PR[GP1:91,2] = PR[GP1:90,2] + 3.452;
   1:L PR[91] 10mm/sec CNT100;
   1:  PR[GP1:91,1] = PR[GP1:90,1] + 66.715;
   1:  PR[GP1:91,2] = PR[GP1:90,2] + 9.248;
   1:L PR[91] 10mm/sec CNT100;
   1:  PR[GP1:91,1] = PR[GP1:90,1] + 64.592;
   1:  PR[GP1:91,2] = PR[GP1:90,2] + 14.983;
   1:L PR[91] 10mm/sec CNT100;
   1:  PR[GP1:91,1] = PR[GP1:90,1] + 63.419;
   1:  PR[GP1:91,2] = PR[GP1:90,2] + 16.961;
   1:L PR[91] 10mm/sec CNT100;
   1:  PR[GP1:91,1] = PR[GP1:90,1] + 59.784;
   1:  PR[GP1:91,2] = PR[GP1:90,2] + 22.603;
   1:L PR[91] 10mm/sec CNT100;
   1:  PR[GP1:91,1] = PR[GP1:90,1] + 54.079;
   1:  PR[GP1:91,2] = PR[GP1:90,2] + 28.157;
   1:L PR[91] 10mm/sec CNT100;
   1:  PR[GP1:91,1] = PR[GP1:90,1] + 54.015;
   1:  PR[GP1:91,2] = PR[GP1:90,2] + 28.216;
   1:L PR[91] 10mm/sec CNT100;
   1:  PR[GP1:91,1] = PR[GP1:90,1] + 47.186;
   1:  PR[GP1:91,2] = PR[GP1:90,2] + 32.500;
   1:L PR[91] 10mm/sec CNT100;
   1:  PR[GP1:91,1] = PR[GP1:90,1] + 46.518;
   1:  PR[GP1:91,2] = PR[GP1:90,2] + 32.792;
   1:L PR[91] 10mm/sec CNT100;
   1:  PR[GP1:91,1] = PR[GP1:90,1] + 39.000;
   1:  PR[GP1:91,2] = PR[GP1:90,2] + 35.536;
   1:L PR[91] 10mm/sec CNT100;
   1:  PR[GP1:91,1] = PR[GP1:90,1] + 31.881;
   1:  PR[GP1:91,2] = PR[GP1:90,2] + 36.545;
   1:L PR[91] 10mm/sec CNT100;
   1:  PR[GP1:91,1] = PR[GP1:90,1] + 29.842;
   1:  PR[GP1:91,2] = PR[GP1:90,2] + 36.734;
   1:L PR[91] 10mm/sec CNT100;
   1:  PR[GP1:91,1] = PR[GP1:90,1] + 22.903;
   1:  PR[GP1:91,2] = PR[GP1:90,2] + 36.273;
   1:L PR[91] 10mm/sec CNT100;
   1:  PR[GP1:91,1] = PR[GP1:90,1] + 20.183;
   1:  PR[GP1:91,2] = PR[GP1:90,2] + 35.631;
   1:L PR[91] 10mm/sec CNT100;
   1:  PR[GP1:91,1] = PR[GP1:90,1] + 13.722;
   1:  PR[GP1:91,2] = PR[GP1:90,2] + 33.773;
   1:L PR[91] 10mm/sec CNT100;
   1:  PR[GP1:91,1] = PR[GP1:90,1] + 8.144;
   1:  PR[GP1:91,2] = PR[GP1:90,2] + 30.769;
   1:L PR[91] 10mm/sec CNT100;
   1:  PR[GP1:91,1] = PR[GP1:90,1] + 1.947;
   1:  PR[GP1:91,2] = PR[GP1:90,2] + 25.729;
   1:L PR[91] 10mm/sec CNT100;
   1:  PR[GP1:91,1] = PR[GP1:90,1] + 1.032;
   1:  PR[GP1:91,2] = PR[GP1:90,2] + 24.922;
   1:L PR[91] 10mm/sec CNT100;
   1:  PR[GP1:91,1] = PR[GP1:90,1] + 0.144;
   1:  PR[GP1:91,2] = PR[GP1:90,2] + 23.840;
   1:L PR[91] 10mm/sec CNT100;
   1:  PR[GP1:91,1] = PR[GP1:90,1] + -0.665;
   1:L PR[91] 10mm/sec CNT100;
   1:  PR[GP1:91,1] = PR[GP1:90,1] + -1.550;
   1:  PR[GP1:91,2] = PR[GP1:90,2] + 24.916;
   1:L PR[91] 10mm/sec CNT100;
   1:  PR[GP1:91,1] = PR[GP1:90,1] + -2.467;
   1:  PR[GP1:91,2] = PR[GP1:90,2] + 25.723;
   1:L PR[91] 10mm/sec CNT100;
   1:  PR[GP1:91,1] = PR[GP1:90,1] + -8.648;
   1:  PR[GP1:91,2] = PR[GP1:90,2] + 30.748;
   1:L PR[91] 10mm/sec CNT100;
   1:  PR[GP1:91,1] = PR[GP1:90,1] + -14.254;
   1:  PR[GP1:91,2] = PR[GP1:90,2] + 33.777;
   1:L PR[91] 10mm/sec CNT100;
   1:  PR[GP1:91,1] = PR[GP1:90,1] + -20.706;
   1:  PR[GP1:91,2] = PR[GP1:90,2] + 35.632;
   1:L PR[91] 10mm/sec CNT100;
   1:  PR[GP1:91,1] = PR[GP1:90,1] + -23.427;
   1:  PR[GP1:91,2] = PR[GP1:90,2] + 36.274;
   1:L PR[91] 10mm/sec CNT100;
   1:  PR[GP1:91,1] = PR[GP1:90,1] + -30.373;
   1:  PR[GP1:91,2] = PR[GP1:90,2] + 36.732;
   1:L PR[91] 10mm/sec CNT100;
   1:  PR[GP1:91,1] = PR[GP1:90,1] + -38.130;
   1:  PR[GP1:91,2] = PR[GP1:90,2] + 35.659;
   1:L PR[91] 10mm/sec CNT100;
   1:  PR[GP1:91,1] = PR[GP1:90,1] + -39.579;
   1:  PR[GP1:91,2] = PR[GP1:90,2] + 35.523;
   1:L PR[91] 10mm/sec CNT100;
   1:  PR[GP1:91,1] = PR[GP1:90,1] + -47.075;
   1:  PR[GP1:91,2] = PR[GP1:90,2] + 32.777;
   1:L PR[91] 10mm/sec CNT100;
   1:  PR[GP1:91,1] = PR[GP1:90,1] + -47.740;
   1:  PR[GP1:91,2] = PR[GP1:90,2] + 32.487;
   1:L PR[91] 10mm/sec CNT100;
   1:  PR[GP1:91,1] = PR[GP1:90,1] + -54.601;
   1:  PR[GP1:91,2] = PR[GP1:90,2] + 28.160;
   1:L PR[91] 10mm/sec CNT100;
   1:  PR[GP1:91,1] = PR[GP1:90,1] + -60.367;
   1:  PR[GP1:91,2] = PR[GP1:90,2] + 22.545;
   1:L PR[91] 10mm/sec CNT100;
   1:  PR[GP1:91,1] = PR[GP1:90,1] + -61.037;
   1:  PR[GP1:91,2] = PR[GP1:90,2] + 21.418;
   1:L PR[91] 10mm/sec CNT100;
   1:  PR[GP1:91,1] = PR[GP1:90,1] + -65.139;
   1:  PR[GP1:91,2] = PR[GP1:90,2] + 14.936;
   1:L PR[91] 10mm/sec CNT100;
   1:  PR[GP1:91,1] = PR[GP1:90,1] + -67.272;
   1:  PR[GP1:91,2] = PR[GP1:90,2] + 9.098;
   1:L PR[91] 10mm/sec CNT100;
   1:  PR[GP1:91,1] = PR[GP1:90,1] + -67.841;
   1:  PR[GP1:91,2] = PR[GP1:90,2] + 5.965;
   1:L PR[91] 10mm/sec CNT100;
   1:  PR[GP1:91,1] = PR[GP1:90,1] + -68.471;
   1:  PR[GP1:91,2] = PR[GP1:90,2] + 0.301;
   1:L PR[91] 10mm/sec CNT100;
   1:  PR[GP1:91,1] = PR[GP1:90,1] + -67.884;
   1:  PR[GP1:91,2] = PR[GP1:90,2] + -2.889;
   1:L PR[91] 10mm/sec CNT100;
   1:  PR[GP1:91,1] = PR[GP1:90,1] + -67.265;
   1:  PR[GP1:91,2] = PR[GP1:90,2] + -8.560;
   1:L PR[91] 10mm/sec CNT100;
   1:  PR[GP1:91,1] = PR[GP1:90,1] + -65.136;
   1:  PR[GP1:91,2] = PR[GP1:90,2] + -14.387;
   1:L PR[91] 10mm/sec CNT100;
   1:  PR[GP1:91,1] = PR[GP1:90,1] + -63.961;
   1:  PR[GP1:91,2] = PR[GP1:90,2] + -16.375;
   1:L PR[91] 10mm/sec CNT100;
   1:  PR[GP1:91,1] = PR[GP1:90,1] + -60.374;
   1:  PR[GP1:91,2] = PR[GP1:90,2] + -21.980;
   1:L PR[91] 10mm/sec CNT100;
   1:  PR[GP1:91,1] = PR[GP1:90,1] + -54.602;
   1:  PR[GP1:91,2] = PR[GP1:90,2] + -27.602;
   1:L PR[91] 10mm/sec CNT100;
   1:  PR[GP1:91,1] = PR[GP1:90,1] + -47.743;
   1:  PR[GP1:91,2] = PR[GP1:90,2] + -31.926;
   1:L PR[91] 10mm/sec CNT100;
   1:  PR[GP1:91,1] = PR[GP1:90,1] + -47.081;
   1:  PR[GP1:91,2] = PR[GP1:90,2] + -32.218;
   1:L PR[91] 10mm/sec CNT100;
   1:  PR[GP1:91,1] = PR[GP1:90,1] + -39.578;
   1:  PR[GP1:91,2] = PR[GP1:90,2] + -34.966;
   1:L PR[91] 10mm/sec CNT100;
   1:  PR[GP1:91,1] = PR[GP1:90,1] + -32.441;
   1:  PR[GP1:91,2] = PR[GP1:90,2] + -35.982;
   1:L PR[91] 10mm/sec CNT100;
   1:  PR[GP1:91,1] = PR[GP1:90,1] + -30.410;
   1:  PR[GP1:91,2] = PR[GP1:90,2] + -36.177;
   1:L PR[91] 10mm/sec CNT100;
   1:  PR[GP1:91,1] = PR[GP1:90,1] + -23.454;
   1:  PR[GP1:91,2] = PR[GP1:90,2] + -35.718;
   1:L PR[91] 10mm/sec CNT100;
   1:  PR[GP1:91,1] = PR[GP1:90,1] + -20.779;
   1:  PR[GP1:91,2] = PR[GP1:90,2] + -35.106;
   1:L PR[91] 10mm/sec CNT100;
   1:  PR[GP1:91,1] = PR[GP1:90,1] + -14.324;
   1:  PR[GP1:91,2] = PR[GP1:90,2] + -33.252;
   1:L PR[91] 10mm/sec CNT100;
   1:  PR[GP1:91,1] = PR[GP1:90,1] + -11.719;
   1:  PR[GP1:91,2] = PR[GP1:90,2] + -31.726;
   1:L PR[91] 10mm/sec CNT100;
   1:  PR[GP1:91,1] = PR[GP1:90,1] + -7.228;
   1:  PR[GP1:91,2] = PR[GP1:90,2] + -29.281;
   1:L PR[91] 10mm/sec CNT100;
   1:  PR[GP1:91,1] = PR[GP1:90,1] + -2.537;
   1:  PR[GP1:91,2] = PR[GP1:90,2] + -25.233;
   1:L PR[91] 10mm/sec CNT100;
   1:  PR[GP1:91,1] = PR[GP1:90,1] + -1.580;
   1:  PR[GP1:91,2] = PR[GP1:90,2] + -24.391;
   1:L PR[91] 10mm/sec CNT100;
   1:  PR[GP1:91,1] = PR[GP1:90,1] + -0.666;
   1:  PR[GP1:91,2] = PR[GP1:90,2] + -23.282;
   1:L PR[91] 10mm/sec CNT100;
   1:  PR[GP1:91,1] = PR[GP1:90,1] + 0.148;
   1:L PR[91] 10mm/sec CNT100;
   1:  PR[GP1:91,1] = PR[GP1:90,1] + 0.835;
   1:  PR[GP1:91,2] = PR[GP1:90,2] + -24.482;
   1:  PR[GP1:91,3] = PR[GP1:90,3] + 52.155;
   1:L PR[91] 10mm/sec CNT100;
   1:  PR[GP1:91,1] = PR[GP1:90,1] + 6.474;
   1:  PR[GP1:91,2] = PR[GP1:90,2] + -29.367;
   1:L PR[91] 10mm/sec CNT100;
   1:  PR[GP1:91,1] = PR[GP1:90,1] + 10.774;
   1:  PR[GP1:91,2] = PR[GP1:90,2] + -31.701;
   1:L PR[91] 10mm/sec CNT100;
   1:  PR[GP1:91,1] = PR[GP1:90,1] + 13.537;
   1:  PR[GP1:91,2] = PR[GP1:90,2] + -33.318;
   1:L PR[91] 10mm/sec CNT100;
   1:  PR[GP1:91,1] = PR[GP1:90,1] + 19.880;
   1:  PR[GP1:91,2] = PR[GP1:90,2] + -35.140;
   1:L PR[91] 10mm/sec CNT100;
   1:  PR[GP1:91,1] = PR[GP1:90,1] + 22.753;
   1:  PR[GP1:91,2] = PR[GP1:90,2] + -35.797;
   1:L PR[91] 10mm/sec CNT100;
   1:  PR[GP1:91,1] = PR[GP1:90,1] + 29.552;
   1:  PR[GP1:91,2] = PR[GP1:90,2] + -36.249;
   1:L PR[91] 10mm/sec CNT100;
   1:  PR[GP1:91,1] = PR[GP1:90,1] + 37.141;
   1:  PR[GP1:91,2] = PR[GP1:90,2] + -35.201;
   1:L PR[91] 10mm/sec CNT100;
   1:  PR[GP1:91,1] = PR[GP1:90,1] + 38.807;
   1:  PR[GP1:91,2] = PR[GP1:90,2] + -35.039;
   1:L PR[91] 10mm/sec CNT100;
   1:  PR[GP1:91,1] = PR[GP1:90,1] + 46.180;
   1:  PR[GP1:91,2] = PR[GP1:90,2] + -32.348;
   1:L PR[91] 10mm/sec CNT100;
   1:  PR[GP1:91,1] = PR[GP1:90,1] + 47.044;
   1:  PR[GP1:91,2] = PR[GP1:90,2] + -31.968;
   1:L PR[91] 10mm/sec CNT100;
   1:  PR[GP1:91,1] = PR[GP1:90,1] + 53.750;
   1:  PR[GP1:91,2] = PR[GP1:90,2] + -27.760;
   1:L PR[91] 10mm/sec CNT100;
   1:  PR[GP1:91,1] = PR[GP1:90,1] + 59.624;
   1:  PR[GP1:91,2] = PR[GP1:90,2] + -22.041;
   1:L PR[91] 10mm/sec CNT100;
   1:  PR[GP1:91,1] = PR[GP1:90,1] + 59.881;
   1:  PR[GP1:91,2] = PR[GP1:90,2] + -21.610;
   1:L PR[91] 10mm/sec CNT100;
   1:  PR[GP1:91,1] = PR[GP1:90,1] + 64.338;
   1:  PR[GP1:91,2] = PR[GP1:90,2] + -14.613;
   1:L PR[91] 10mm/sec CNT100;
   1:  PR[GP1:91,1] = PR[GP1:90,1] + 66.619;
   1:  PR[GP1:91,2] = PR[GP1:90,2] + -8.452;
   1:L PR[91] 10mm/sec CNT100;
   1:  PR[GP1:91,1] = PR[GP1:90,1] + 67.065;
   1:  PR[GP1:91,2] = PR[GP1:90,2] + -5.989;
   1:L PR[91] 10mm/sec CNT100;
   1:  PR[GP1:91,1] = PR[GP1:90,1] + 67.771;
   1:  PR[GP1:91,2] = PR[GP1:90,2] + 0.258;
   1:L PR[91] 10mm/sec CNT100;
   1:  PR[GP1:91,1] = PR[GP1:90,1] + 67.300;
   1:  PR[GP1:91,2] = PR[GP1:90,2] + 2.819;
   1:L PR[91] 10mm/sec CNT100;
   1:  PR[GP1:91,1] = PR[GP1:90,1] + 66.612;
   1:  PR[GP1:91,2] = PR[GP1:90,2] + 9.030;
   1:L PR[91] 10mm/sec CNT100;
   1:  PR[GP1:91,1] = PR[GP1:90,1] + 64.334;
   1:  PR[GP1:91,2] = PR[GP1:90,2] + 15.181;
   1:L PR[91] 10mm/sec CNT100;
   1:  PR[GP1:91,1] = PR[GP1:90,1] + 63.496;
   1:  PR[GP1:91,2] = PR[GP1:90,2] + 16.596;
   1:L PR[91] 10mm/sec CNT100;
   1:  PR[GP1:91,1] = PR[GP1:90,1] + 59.631;
   1:  PR[GP1:91,2] = PR[GP1:90,2] + 22.592;
   1:L PR[91] 10mm/sec CNT100;
   1:  PR[GP1:91,1] = PR[GP1:90,1] + 53.981;
   1:  PR[GP1:91,2] = PR[GP1:90,2] + 28.112;
   1:L PR[91] 10mm/sec CNT100;
   1:  PR[GP1:91,1] = PR[GP1:90,1] + 53.758;
   1:  PR[GP1:91,2] = PR[GP1:90,2] + 28.314;
   1:L PR[91] 10mm/sec CNT100;
   1:  PR[GP1:91,1] = PR[GP1:90,1] + 47.039;
   1:  PR[GP1:91,2] = PR[GP1:90,2] + 32.529;
   1:L PR[91] 10mm/sec CNT100;
   1:  PR[GP1:91,1] = PR[GP1:90,1] + 46.172;
   1:  PR[GP1:91,2] = PR[GP1:90,2] + 32.908;
   1:L PR[91] 10mm/sec CNT100;
   1:  PR[GP1:91,1] = PR[GP1:90,1] + 38.780;
   1:  PR[GP1:91,2] = PR[GP1:90,2] + 35.606;
   1:L PR[91] 10mm/sec CNT100;
   1:  PR[GP1:91,1] = PR[GP1:90,1] + 31.782;
   1:  PR[GP1:91,2] = PR[GP1:90,2] + 36.598;
   1:L PR[91] 10mm/sec CNT100;
   1:  PR[GP1:91,1] = PR[GP1:90,1] + 29.540;
   1:  PR[GP1:91,2] = PR[GP1:90,2] + 36.806;
   1:L PR[91] 10mm/sec CNT100;
   1:  PR[GP1:91,1] = PR[GP1:90,1] + 22.724;
   1:  PR[GP1:91,2] = PR[GP1:90,2] + 36.354;
   1:L PR[91] 10mm/sec CNT100;
   1:  PR[GP1:91,1] = PR[GP1:90,1] + 19.802;
   1:  PR[GP1:91,2] = PR[GP1:90,2] + 35.663;
   1:L PR[91] 10mm/sec CNT100;
   1:  PR[GP1:91,1] = PR[GP1:90,1] + 13.464;
   1:  PR[GP1:91,2] = PR[GP1:90,2] + 33.841;
   1:L PR[91] 10mm/sec CNT100;
   1:  PR[GP1:91,1] = PR[GP1:90,1] + 7.971;
   1:  PR[GP1:91,2] = PR[GP1:90,2] + 30.883;
   1:L PR[91] 10mm/sec CNT100;
   1:  PR[GP1:91,1] = PR[GP1:90,1] + 1.463;
   1:  PR[GP1:91,2] = PR[GP1:90,2] + 25.589;
   1:L PR[91] 10mm/sec CNT100;
   1:  PR[GP1:91,1] = PR[GP1:90,1] + 0.803;
   1:  PR[GP1:91,2] = PR[GP1:90,2] + 25.008;
   1:L PR[91] 10mm/sec CNT100;
   1:  PR[GP1:91,1] = PR[GP1:90,1] + 0.112;
   1:  PR[GP1:91,2] = PR[GP1:90,2] + 24.165;
   1:L PR[91] 10mm/sec CNT100;
   1:  PR[GP1:91,1] = PR[GP1:90,1] + -0.633;
   1:L PR[91] 10mm/sec CNT100;
   1:  PR[GP1:91,1] = PR[GP1:90,1] + -1.323;
   1:  PR[GP1:91,2] = PR[GP1:90,2] + 25.003;
   1:L PR[91] 10mm/sec CNT100;
   1:  PR[GP1:91,1] = PR[GP1:90,1] + -1.984;
   1:  PR[GP1:91,2] = PR[GP1:90,2] + 25.585;
   1:L PR[91] 10mm/sec CNT100;
   1:  PR[GP1:91,1] = PR[GP1:90,1] + -8.475;
   1:  PR[GP1:91,2] = PR[GP1:90,2] + 30.862;
   1:L PR[91] 10mm/sec CNT100;
   1:  PR[GP1:91,1] = PR[GP1:90,1] + -13.995;
   1:  PR[GP1:91,2] = PR[GP1:90,2] + 33.844;
   1:L PR[91] 10mm/sec CNT100;
   1:  PR[GP1:91,1] = PR[GP1:90,1] + -20.325;
   1:  PR[GP1:91,2] = PR[GP1:90,2] + 35.664;
   1:L PR[91] 10mm/sec CNT100;
   1:  PR[GP1:91,1] = PR[GP1:90,1] + -23.248;
   1:  PR[GP1:91,2] = PR[GP1:90,2] + 36.354;
   1:L PR[91] 10mm/sec CNT100;
   1:  PR[GP1:91,1] = PR[GP1:90,1] + -30.071;
   1:  PR[GP1:91,2] = PR[GP1:90,2] + 36.804;
   1:L PR[91] 10mm/sec CNT100;
   1:  PR[GP1:91,1] = PR[GP1:90,1] + -37.691;
   1:  PR[GP1:91,2] = PR[GP1:90,2] + 35.750;
   1:L PR[91] 10mm/sec CNT100;
   1:  PR[GP1:91,1] = PR[GP1:90,1] + -39.359;
   1:  PR[GP1:91,2] = PR[GP1:90,2] + 35.593;
   1:L PR[91] 10mm/sec CNT100;
   1:  PR[GP1:91,1] = PR[GP1:90,1] + -46.728;
   1:  PR[GP1:91,2] = PR[GP1:90,2] + 32.894;
   1:L PR[91] 10mm/sec CNT100;
   1:  PR[GP1:91,1] = PR[GP1:90,1] + -47.593;
   1:  PR[GP1:91,2] = PR[GP1:90,2] + 32.516;
   1:L PR[91] 10mm/sec CNT100;
   1:  PR[GP1:91,1] = PR[GP1:90,1] + -54.343;
   1:  PR[GP1:91,2] = PR[GP1:90,2] + 28.260;
   1:L PR[91] 10mm/sec CNT100;
   1:  PR[GP1:91,1] = PR[GP1:90,1] + -60.219;
   1:  PR[GP1:91,2] = PR[GP1:90,2] + 22.529;
   1:L PR[91] 10mm/sec CNT100;
   1:  PR[GP1:91,1] = PR[GP1:90,1] + -60.487;
   1:  PR[GP1:91,2] = PR[GP1:90,2] + 22.078;
   1:L PR[91] 10mm/sec CNT100;
   1:  PR[GP1:91,1] = PR[GP1:90,1] + -64.883;
   1:  PR[GP1:91,2] = PR[GP1:90,2] + 15.133;
   1:L PR[91] 10mm/sec CNT100;
   1:  PR[GP1:91,1] = PR[GP1:90,1] + -67.171;
   1:  PR[GP1:91,2] = PR[GP1:90,2] + 8.873;
   1:L PR[91] 10mm/sec CNT100;
   1:  PR[GP1:91,1] = PR[GP1:90,1] + -67.618;
   1:  PR[GP1:91,2] = PR[GP1:90,2] + 6.409;
   1:L PR[91] 10mm/sec CNT100;
   1:  PR[GP1:91,1] = PR[GP1:90,1] + -68.297;
   1:  PR[GP1:91,2] = PR[GP1:90,2] + 0.301;
   1:L PR[91] 10mm/sec CNT100;
   1:  PR[GP1:91,1] = PR[GP1:90,1] + -67.826;
   1:  PR[GP1:91,2] = PR[GP1:90,2] + -2.257;
   1:L PR[91] 10mm/sec CNT100;
   1:  PR[GP1:91,1] = PR[GP1:90,1] + -67.163;
   1:  PR[GP1:91,2] = PR[GP1:90,2] + -8.335;
   1:L PR[91] 10mm/sec CNT100;
   1:  PR[GP1:91,1] = PR[GP1:90,1] + -64.879;
   1:  PR[GP1:91,2] = PR[GP1:90,2] + -14.584;
   1:L PR[91] 10mm/sec CNT100;
   1:  PR[GP1:91,1] = PR[GP1:90,1] + -64.039;
   1:  PR[GP1:91,2] = PR[GP1:90,2] + -16.007;
   1:L PR[91] 10mm/sec CNT100;
   1:  PR[GP1:91,1] = PR[GP1:90,1] + -60.226;
   1:  PR[GP1:91,2] = PR[GP1:90,2] + -21.964;
   1:L PR[91] 10mm/sec CNT100;
   1:  PR[GP1:91,1] = PR[GP1:90,1] + -54.573;
   1:  PR[GP1:91,2] = PR[GP1:90,2] + -27.496;
   1:L PR[91] 10mm/sec CNT100;
   1:  PR[GP1:91,1] = PR[GP1:90,1] + -54.354;
   1:  PR[GP1:91,2] = PR[GP1:90,2] + -27.695;
   1:L PR[91] 10mm/sec CNT100;
   1:  PR[GP1:91,1] = PR[GP1:90,1] + -47.598;
   1:  PR[GP1:91,2] = PR[GP1:90,2] + -31.955;
   1:L PR[91] 10mm/sec CNT100;
   1:  PR[GP1:91,1] = PR[GP1:90,1] + -46.737;
   1:  PR[GP1:91,2] = PR[GP1:90,2] + -32.334;
   1:L PR[91] 10mm/sec CNT100;
   1:  PR[GP1:91,1] = PR[GP1:90,1] + -39.359;
   1:  PR[GP1:91,2] = PR[GP1:90,2] + -35.036;
   1:L PR[91] 10mm/sec CNT100;
   1:  PR[GP1:91,1] = PR[GP1:90,1] + -32.343;
   1:  PR[GP1:91,2] = PR[GP1:90,2] + -36.034;
   1:L PR[91] 10mm/sec CNT100;
   1:  PR[GP1:91,1] = PR[GP1:90,1] + -30.109;
   1:  PR[GP1:91,2] = PR[GP1:90,2] + -36.249;
   1:L PR[91] 10mm/sec CNT100;
   1:  PR[GP1:91,1] = PR[GP1:90,1] + -23.277;
   1:  PR[GP1:91,2] = PR[GP1:90,2] + -35.798;
   1:L PR[91] 10mm/sec CNT100;
   1:  PR[GP1:91,1] = PR[GP1:90,1] + -20.403;
   1:  PR[GP1:91,2] = PR[GP1:90,2] + -35.140;
   1:L PR[91] 10mm/sec CNT100;
   1:  PR[GP1:91,1] = PR[GP1:90,1] + -14.069;
   1:  PR[GP1:91,2] = PR[GP1:90,2] + -33.321;
   1:L PR[91] 10mm/sec CNT100;
   1:  PR[GP1:91,1] = PR[GP1:90,1] + -11.308;
   1:  PR[GP1:91,2] = PR[GP1:90,2] + -31.704;
   1:L PR[91] 10mm/sec CNT100;
   1:  PR[GP1:91,1] = PR[GP1:90,1] + -6.985;
   1:  PR[GP1:91,2] = PR[GP1:90,2] + -29.351;
   1:L PR[91] 10mm/sec CNT100;
   1:  PR[GP1:91,1] = PR[GP1:90,1] + -1.352;
   1:  PR[GP1:91,2] = PR[GP1:90,2] + -24.477;
   1:L PR[91] 10mm/sec CNT100;
   1:  PR[GP1:91,1] = PR[GP1:90,1] + -0.635;
   1:  PR[GP1:91,2] = PR[GP1:90,2] + -23.607;
   1:L PR[91] 10mm/sec CNT100;
   1:  PR[GP1:91,1] = PR[GP1:90,1] + 0.116;
   1:L PR[91] 10mm/sec CNT100;
   1:  PR[GP1:91,1] = PR[GP1:90,1] + 0.608;
   1:  PR[GP1:91,2] = PR[GP1:90,2] + -24.569;
   1:  PR[GP1:91,3] = PR[GP1:90,3] + 52.765;
   1:L PR[91] 10mm/sec CNT100;
   1:  PR[GP1:91,1] = PR[GP1:90,1] + 6.230;
   1:  PR[GP1:91,2] = PR[GP1:90,2] + -29.436;
   1:L PR[91] 10mm/sec CNT100;
   1:  PR[GP1:91,1] = PR[GP1:90,1] + 10.363;
   1:  PR[GP1:91,2] = PR[GP1:90,2] + -31.679;
   1:L PR[91] 10mm/sec CNT100;
   1:  PR[GP1:91,1] = PR[GP1:90,1] + 13.282;
   1:  PR[GP1:91,2] = PR[GP1:90,2] + -33.388;
   1:L PR[91] 10mm/sec CNT100;
   1:  PR[GP1:91,1] = PR[GP1:90,1] + 19.504;
   1:  PR[GP1:91,2] = PR[GP1:90,2] + -35.174;
   1:L PR[91] 10mm/sec CNT100;
   1:  PR[GP1:91,1] = PR[GP1:90,1] + 22.577;
   1:  PR[GP1:91,2] = PR[GP1:90,2] + -35.877;
   1:L PR[91] 10mm/sec CNT100;
   1:  PR[GP1:91,1] = PR[GP1:90,1] + 29.252;
   1:  PR[GP1:91,2] = PR[GP1:90,2] + -36.321;
   1:L PR[91] 10mm/sec CNT100;
   1:  PR[GP1:91,1] = PR[GP1:90,1] + 36.705;
   1:  PR[GP1:91,2] = PR[GP1:90,2] + -35.292;
   1:L PR[91] 10mm/sec CNT100;
   1:  PR[GP1:91,1] = PR[GP1:90,1] + 38.589;
   1:  PR[GP1:91,2] = PR[GP1:90,2] + -35.109;
   1:L PR[91] 10mm/sec CNT100;
   1:  PR[GP1:91,1] = PR[GP1:90,1] + 45.836;
   1:  PR[GP1:91,2] = PR[GP1:90,2] + -32.464;
   1:L PR[91] 10mm/sec CNT100;
   1:  PR[GP1:91,1] = PR[GP1:90,1] + 46.899;
   1:  PR[GP1:91,2] = PR[GP1:90,2] + -31.997;
   1:L PR[91] 10mm/sec CNT100;
   1:  PR[GP1:91,1] = PR[GP1:90,1] + 53.495;
   1:  PR[GP1:91,2] = PR[GP1:90,2] + -27.858;
   1:L PR[91] 10mm/sec CNT100;
   1:  PR[GP1:91,1] = PR[GP1:90,1] + 59.469;
   1:  PR[GP1:91,2] = PR[GP1:90,2] + -22.038;
   1:L PR[91] 10mm/sec CNT100;
   1:  PR[GP1:91,1] = PR[GP1:90,1] + 64.080;
   1:  PR[GP1:91,2] = PR[GP1:90,2] + -14.811;
   1:L PR[91] 10mm/sec CNT100;
   1:  PR[GP1:91,1] = PR[GP1:90,1] + 66.516;
   1:  PR[GP1:91,2] = PR[GP1:90,2] + -8.235;
   1:L PR[91] 10mm/sec CNT100;
   1:  PR[GP1:91,1] = PR[GP1:90,1] + 66.840;
   1:  PR[GP1:91,2] = PR[GP1:90,2] + -6.443;
   1:L PR[91] 10mm/sec CNT100;
   1:  PR[GP1:91,1] = PR[GP1:90,1] + 67.597;
   1:  PR[GP1:91,2] = PR[GP1:90,2] + 0.258;
   1:L PR[91] 10mm/sec CNT100;
   1:  PR[GP1:91,1] = PR[GP1:90,1] + 67.242;
   1:  PR[GP1:91,2] = PR[GP1:90,2] + 2.187;
   1:L PR[91] 10mm/sec CNT100;
   1:  PR[GP1:91,1] = PR[GP1:90,1] + 66.508;
   1:  PR[GP1:91,2] = PR[GP1:90,2] + 8.812;
   1:L PR[91] 10mm/sec CNT100;
   1:  PR[GP1:91,1] = PR[GP1:90,1] + 64.077;
   1:  PR[GP1:91,2] = PR[GP1:90,2] + 15.379;
   1:L PR[91] 10mm/sec CNT100;
   1:  PR[GP1:91,1] = PR[GP1:90,1] + 63.572;
   1:  PR[GP1:91,2] = PR[GP1:90,2] + 16.230;
   1:L PR[91] 10mm/sec CNT100;
   1:  PR[GP1:91,1] = PR[GP1:90,1] + 59.470;
   1:  PR[GP1:91,2] = PR[GP1:90,2] + 22.596;
   1:L PR[91] 10mm/sec CNT100;
   1:  PR[GP1:91,1] = PR[GP1:90,1] + 53.884;
   1:  PR[GP1:91,2] = PR[GP1:90,2] + 28.066;
   1:L PR[91] 10mm/sec CNT100;
   1:  PR[GP1:91,1] = PR[GP1:90,1] + 53.501;
   1:  PR[GP1:91,2] = PR[GP1:90,2] + 28.412;
   1:L PR[91] 10mm/sec CNT100;
   1:  PR[GP1:91,1] = PR[GP1:90,1] + 46.893;
   1:  PR[GP1:91,2] = PR[GP1:90,2] + 32.558;
   1:L PR[91] 10mm/sec CNT100;
   1:  PR[GP1:91,1] = PR[GP1:90,1] + 45.826;
   1:  PR[GP1:91,2] = PR[GP1:90,2] + 33.025;
   1:L PR[91] 10mm/sec CNT100;
   1:  PR[GP1:91,1] = PR[GP1:90,1] + 38.561;
   1:  PR[GP1:91,2] = PR[GP1:90,2] + 35.676;
   1:L PR[91] 10mm/sec CNT100;
   1:  PR[GP1:91,1] = PR[GP1:90,1] + 31.683;
   1:  PR[GP1:91,2] = PR[GP1:90,2] + 36.651;
   1:L PR[91] 10mm/sec CNT100;
   1:  PR[GP1:91,1] = PR[GP1:90,1] + 29.237;
   1:  PR[GP1:91,2] = PR[GP1:90,2] + 36.878;
   1:L PR[91] 10mm/sec CNT100;
   1:  PR[GP1:91,1] = PR[GP1:90,1] + 22.545;
   1:  PR[GP1:91,2] = PR[GP1:90,2] + 36.434;
   1:L PR[91] 10mm/sec CNT100;
   1:  PR[GP1:91,1] = PR[GP1:90,1] + 19.422;
   1:  PR[GP1:91,2] = PR[GP1:90,2] + 35.696;
   1:L PR[91] 10mm/sec CNT100;
   1:  PR[GP1:91,1] = PR[GP1:90,1] + 13.206;
   1:  PR[GP1:91,2] = PR[GP1:90,2] + 33.909;
   1:L PR[91] 10mm/sec CNT100;
   1:  PR[GP1:91,1] = PR[GP1:90,1] + 7.798;
   1:  PR[GP1:91,2] = PR[GP1:90,2] + 30.997;
   1:L PR[91] 10mm/sec CNT100;
   1:  PR[GP1:91,1] = PR[GP1:90,1] + 0.978;
   1:  PR[GP1:91,2] = PR[GP1:90,2] + 25.449;
   1:L PR[91] 10mm/sec CNT100;
   1:  PR[GP1:91,1] = PR[GP1:90,1] + 0.574;
   1:  PR[GP1:91,2] = PR[GP1:90,2] + 25.093;
   1:L PR[91] 10mm/sec CNT100;
   1:  PR[GP1:91,1] = PR[GP1:90,1] + 0.079;
   1:  PR[GP1:91,2] = PR[GP1:90,2] + 24.490;
   1:L PR[91] 10mm/sec CNT100;
   1:  PR[GP1:91,1] = PR[GP1:90,1] + -0.602;
   1:L PR[91] 10mm/sec CNT100;
   1:  PR[GP1:91,1] = PR[GP1:90,1] + -1.096;
   1:  PR[GP1:91,2] = PR[GP1:90,2] + 25.090;
   1:L PR[91] 10mm/sec CNT100;
   1:  PR[GP1:91,1] = PR[GP1:90,1] + -1.501;
   1:  PR[GP1:91,2] = PR[GP1:90,2] + 25.447;
   1:L PR[91] 10mm/sec CNT100;
   1:  PR[GP1:91,1] = PR[GP1:90,1] + -8.303;
   1:  PR[GP1:91,2] = PR[GP1:90,2] + 30.977;
   1:L PR[91] 10mm/sec CNT100;
   1:  PR[GP1:91,1] = PR[GP1:90,1] + -13.737;
   1:  PR[GP1:91,2] = PR[GP1:90,2] + 33.912;
   1:L PR[91] 10mm/sec CNT100;
   1:  PR[GP1:91,1] = PR[GP1:90,1] + -19.945;
   1:  PR[GP1:91,2] = PR[GP1:90,2] + 35.696;
   1:L PR[91] 10mm/sec CNT100;
   1:  PR[GP1:91,1] = PR[GP1:90,1] + -23.069;
   1:  PR[GP1:91,2] = PR[GP1:90,2] + 36.434;
   1:L PR[91] 10mm/sec CNT100;
   1:  PR[GP1:91,1] = PR[GP1:90,1] + -29.768;
   1:  PR[GP1:91,2] = PR[GP1:90,2] + 36.876;
   1:L PR[91] 10mm/sec CNT100;
   1:  PR[GP1:91,1] = PR[GP1:90,1] + -37.252;
   1:  PR[GP1:91,2] = PR[GP1:90,2] + 35.840;
   1:L PR[91] 10mm/sec CNT100;
   1:  PR[GP1:91,1] = PR[GP1:90,1] + -39.139;
   1:  PR[GP1:91,2] = PR[GP1:90,2] + 35.663;
   1:L PR[91] 10mm/sec CNT100;
   1:  PR[GP1:91,1] = PR[GP1:90,1] + -46.382;
   1:  PR[GP1:91,2] = PR[GP1:90,2] + 33.010;
   1:L PR[91] 10mm/sec CNT100;
   1:  PR[GP1:91,1] = PR[GP1:90,1] + -47.446;
   1:  PR[GP1:91,2] = PR[GP1:90,2] + 32.545;
   1:L PR[91] 10mm/sec CNT100;
   1:  PR[GP1:91,1] = PR[GP1:90,1] + -54.085;
   1:  PR[GP1:91,2] = PR[GP1:90,2] + 28.359;
   1:L PR[91] 10mm/sec CNT100;
   1:  PR[GP1:91,1] = PR[GP1:90,1] + -60.068;
   1:  PR[GP1:91,2] = PR[GP1:90,2] + 22.522;
   1:L PR[91] 10mm/sec CNT100;
   1:  PR[GP1:91,1] = PR[GP1:90,1] + -64.627;
   1:  PR[GP1:91,2] = PR[GP1:90,2] + 15.330;
   1:L PR[91] 10mm/sec CNT100;
   1:  PR[GP1:91,1] = PR[GP1:90,1] + -67.069;
   1:  PR[GP1:91,2] = PR[GP1:90,2] + 8.648;
   1:L PR[91] 10mm/sec CNT100;
   1:  PR[GP1:91,1] = PR[GP1:90,1] + -67.394;
   1:  PR[GP1:91,2] = PR[GP1:90,2] + 6.852;
   1:L PR[91] 10mm/sec CNT100;
   1:  PR[GP1:91,1] = PR[GP1:90,1] + -68.123;
   1:  PR[GP1:91,2] = PR[GP1:90,2] + 0.301;
   1:L PR[91] 10mm/sec CNT100;
   1:  PR[GP1:91,1] = PR[GP1:90,1] + -67.768;
   1:  PR[GP1:91,2] = PR[GP1:90,2] + -1.625;
   1:L PR[91] 10mm/sec CNT100;
   1:  PR[GP1:91,1] = PR[GP1:90,1] + -67.061;
   1:  PR[GP1:91,2] = PR[GP1:90,2] + -8.110;
   1:L PR[91] 10mm/sec CNT100;
   1:  PR[GP1:91,1] = PR[GP1:90,1] + -64.623;
   1:  PR[GP1:91,2] = PR[GP1:90,2] + -14.781;
   1:L PR[91] 10mm/sec CNT100;
   1:  PR[GP1:91,1] = PR[GP1:90,1] + -64.116;
   1:  PR[GP1:91,2] = PR[GP1:90,2] + -15.639;
   1:L PR[91] 10mm/sec CNT100;
   1:  PR[GP1:91,1] = PR[GP1:90,1] + -60.068;
   1:  PR[GP1:91,2] = PR[GP1:90,2] + -21.963;
   1:L PR[91] 10mm/sec CNT100;
   1:  PR[GP1:91,1] = PR[GP1:90,1] + -54.475;
   1:  PR[GP1:91,2] = PR[GP1:90,2] + -27.451;
   1:L PR[91] 10mm/sec CNT100;
   1:  PR[GP1:91,1] = PR[GP1:90,1] + -54.097;
   1:  PR[GP1:91,2] = PR[GP1:90,2] + -27.793;
   1:L PR[91] 10mm/sec CNT100;
   1:  PR[GP1:91,1] = PR[GP1:90,1] + -47.452;
   1:  PR[GP1:91,2] = PR[GP1:90,2] + -31.983;
   1:L PR[91] 10mm/sec CNT100;
   1:  PR[GP1:91,1] = PR[GP1:90,1] + -46.392;
   1:  PR[GP1:91,2] = PR[GP1:90,2] + -32.450;
   1:L PR[91] 10mm/sec CNT100;
   1:  PR[GP1:91,1] = PR[GP1:90,1] + -39.141;
   1:  PR[GP1:91,2] = PR[GP1:90,2] + -35.106;
   1:L PR[91] 10mm/sec CNT100;
   1:  PR[GP1:91,1] = PR[GP1:90,1] + -32.245;
   1:  PR[GP1:91,2] = PR[GP1:90,2] + -36.087;
   1:L PR[91] 10mm/sec CNT100;
